LIN {X 0,Y 688.644,Z 762.06,A -85,B 0,C 180,E1 4140.007,E2 4140.007} C_VEL
LIN {X 0,Y 688.645,Z 762.06,A -85,B 0,C 180,E1 4145.042,E2 4145.042} C_VEL
LIN {X 0,Y 688.471,Z 762.06,A -85,B 0,C 180,E1 4150.119,E2 4150.119} C_VEL
LIN {X 0,Y 688.438,Z 762.06,A -85,B 0,C 180,E1 4155.277,E2 4155.277} C_VEL
LIN {X 0,Y 688.385,Z 762.06,A -85,B 0,C 180,E1 4160.05,E2 4160.05} C_VEL
LIN {X 0,Y 687.119,Z 762.06,A -85,B 0,C 180,E1 4160.769,E2 4160.769} C_VEL
LIN {X 0,Y 680.471,Z 762.06,A -85,B 0,C 180,E1 4162.723,E2 4162.723} C_VEL
LIN {X 0,Y 680.377,Z 762.06,A -85,B 0,C 180,E1 4162.908,E2 4162.908} C_VEL
LIN {X 0,Y 680.412,Z 762.06,A -85,B 0,C 180,E1 4167.804,E2 4167.804} C_VEL
LIN {X 0,Y 680.284,Z 762.06,A -85,B 0,C 180,E1 4172.424,E2 4172.424} C_VEL
LIN {X 0,Y 680.225,Z 762.06,A -85,B 0,C 180,E1 4176.894,E2 4176.894} C_VEL
LIN {X 0,Y 680.38,Z 762.06,A -85,B 0,C 180,E1 4182.867,E2 4182.867} C_VEL
LIN {X 0,Y 680.225,Z 762.06,A -85,B 0,C 180,E1 4188.271,E2 4188.271} C_VEL
LIN {X 0,Y 685.455,Z 772.734,A -85,B 0,C 180,E1 4188.863,E2 4188.863} C_VEL
LIN {X 0,Y 698.064,Z 795.344,A -85,B 0,C 180,E1 4190.059,E2 4190.059} C_VEL
LIN {X 0,Y 697.442,Z 854.76,A -85,B 0,C 180,E1 4190.981,E2 4190.981} C_VEL
LIN {X 0,Y 695.603,Z 898.868,A -85,B 0,C 180,E1 4192.105,E2 4192.105} C_VEL
LIN {X 0,Y 693.258,Z 948.265,A -85,B 0,C 180,E1 4193.947,E2 4193.947} C_VEL
LIN {X 0,Y 690.751,Z 992.677,A -85,B 0,C 180,E1 4196.173,E2 4196.173} C_VEL
LIN {X 0,Y 688.172,Z 1037.406,A -85,B 0,C 180,E1 4199.062,E2 4199.062} C_VEL
LIN {X 0,Y 685.781,Z 1076.683,A -85,B 0,C 180,E1 4202.265,E2 4202.265} C_VEL
LIN {X 0,Y 683.938,Z 1110.79,A -85,B 0,C 180,E1 4205.7,E2 4205.7} C_VEL
LIN {X 0,Y 682.434,Z 1142.324,A -85,B 0,C 180,E1 4209.682,E2 4209.682} C_VEL
LIN {X 0,Y 681.538,Z 1166.468,A -85,B 0,C 180,E1 4213.578,E2 4213.578} C_VEL
LIN {X 0,Y 681.033,Z 1185.03,A -85,B 0,C 180,E1 4217.501,E2 4217.501} C_VEL
LIN {X 0,Y 680.865,Z 1197.33,A -85,B 0,C 180,E1 4221.062,E2 4221.062} C_VEL
LIN {X 0,Y 680.767,Z 1205.91,A -85,B 0,C 180,E1 4224.905,E2 4224.905} C_VEL
LIN {X 0,Y 680.672,Z 1209.668,A -85,B 0,C 180,E1 4228.727,E2 4228.727} C_VEL
LIN {X 0,Y 680.871,Z 1208.953,A -85,B 0,C 180,E1 4232.543,E2 4232.543} C_VEL
LIN {X 0,Y 680.861,Z 1203.571,A -85,B 0,C 180,E1 4236.371,E2 4236.371} C_VEL
LIN {X 0,Y 681.018,Z 1192.319,A -85,B 0,C 180,E1 4240.547,E2 4240.547} C_VEL
LIN {X 0,Y 681.312,Z 1175.162,A -85,B 0,C 180,E1 4244.725,E2 4244.725} C_VEL
LIN {X 0,Y 682.005,Z 1153.941,A -85,B 0,C 180,E1 4248.572,E2 4248.572} C_VEL
LIN {X 0,Y 683.15,Z 1126.486,A -85,B 0,C 180,E1 4252.43,E2 4252.43} C_VEL
LIN {X 0,Y 684.773,Z 1094.478,A -85,B 0,C 180,E1 4256.038,E2 4256.038} C_VEL
LIN {X 0,Y 687.044,Z 1055.156,A -85,B 0,C 180,E1 4259.585,E2 4259.585} C_VEL
LIN {X 0,Y 689.594,Z 1013.392,A -85,B 0,C 180,E1 4262.572,E2 4262.572} C_VEL
LIN {X 0,Y 692.183,Z 970.786,A -85,B 0,C 180,E1 4264.995,E2 4264.995} C_VEL
LIN {X 0,Y 694.562,Z 925.309,A -85,B 0,C 180,E1 4266.975,E2 4266.975} C_VEL
LIN {X 0,Y 696.481,Z 879.014,A -85,B 0,C 180,E1 4268.46,E2 4268.46} C_VEL
LIN {X 0,Y 697.908,Z 831.825,A -85,B 0,C 180,E1 4269.439,E2 4269.439} C_VEL
LIN {X 0,Y 697.724,Z 794.961,A -85,B 0,C 180,E1 4269.969,E2 4269.969} C_VEL
LIN {X 0,Y 680.46,Z 763.676,A -85,B 0,C 180,E1 4271.63,E2 4271.63} C_VEL
LIN {X 0,Y 680.306,Z 762.06,A -85,B 0,C 180,E1 4271.725,E2 4271.725} C_VEL
LIN {X 0,Y 680.274,Z 762.06,A -85,B 0,C 180,E1 4276.476,E2 4276.476} C_VEL
LIN {X 0,Y 680.206,Z 762.06,A -85,B 0,C 180,E1 4281.532,E2 4281.532} C_VEL
LIN {X 0,Y 680.178,Z 762.06,A -85,B 0,C 180,E1 4286.257,E2 4286.257} C_VEL
LIN {X 0,Y 680.205,Z 762.06,A -85,B 0,C 180,E1 4290.738,E2 4290.738} C_VEL
LIN {X 0,Y 680.287,Z 762.06,A -85,B 0,C 180,E1 4295.604,E2 4295.604} C_VEL
LIN {X 0,Y 680.322,Z 762.06,A -85,B 0,C 180,E1 4300.533,E2 4300.533} C_VEL
LIN {X 0,Y 680.504,Z 762.06,A -85,B 0,C 180,E1 4304.54,E2 4304.54} C_VEL
LIN {X 0,Y 680.545,Z 762.06,A -85,B 0,C 180,E1 4309.762,E2 4309.762} C_VEL
LIN {X 0,Y 680.769,Z 762.06,A -85,B 0,C 180,E1 4314.899,E2 4314.899} C_VEL
LIN {X 0,Y 680.714,Z 762.06,A -85,B 0,C 180,E1 4319.993,E2 4319.993} C_VEL
LIN {X 0,Y 680.699,Z 762.06,A -85,B 0,C 180,E1 4325.086,E2 4325.086} C_VEL
LIN {X 0,Y 680.588,Z 762.06,A -85,B 0,C 180,E1 4330.223,E2 4330.223} C_VEL
LIN {X 0,Y 680.249,Z 762.06,A -85,B 0,C 180,E1 4335.451,E2 4335.451} C_VEL
LIN {X 0,Y 680.284,Z 762.06,A -85,B 0,C 180,E1 4341.103,E2 4341.103} C_VEL
LIN {X 0,Y 680.228,Z 762.06,A -85,B 0,C 180,E1 4346.366,E2 4346.366} C_VEL
LIN {X 0,Y 680.227,Z 762.06,A -85,B 0,C 180,E1 4350.714,E2 4350.714} C_VEL
LIN {X 0,Y 680.253,Z 762.06,A -85,B 0,C 180,E1 4355.265,E2 4355.265} C_VEL
LIN {X 0,Y 680.097,Z 762.06,A -85,B 0,C 180,E1 4360.101,E2 4360.101} C_VEL
LIN {X 0,Y 680.121,Z 762.06,A -85,B 0,C 180,E1 4365.297,E2 4365.297} C_VEL
LIN {X 0,Y 680.444,Z 762.06,A -85,B 0,C 180,E1 4368.694,E2 4368.694} C_VEL
LIN {X 0,Y 684.939,Z 771.765,A -85,B 0,C 180,E1 4369.176,E2 4369.176} C_VEL
LIN {X 0,Y 698.059,Z 795.739,A -85,B 0,C 180,E1 4370.431,E2 4370.431} C_VEL
LIN {X 0,Y 696.879,Z 840.886,A -85,B 0,C 180,E1 4371.297,E2 4371.297} C_VEL
LIN {X 0,Y 694.891,Z 887.195,A -85,B 0,C 180,E1 4372.674,E2 4372.674} C_VEL
LIN {X 0,Y 692.53,Z 933.533,A -85,B 0,C 180,E1 4374.61,E2 4374.61} C_VEL
LIN {X 0,Y 689.958,Z 977.454,A -85,B 0,C 180,E1 4377.004,E2 4377.004} C_VEL
LIN {X 0,Y 687.283,Z 1021.111,A -85,B 0,C 180,E1 4380.054,E2 4380.054} C_VEL
LIN {X 0,Y 685.096,Z 1057.631,A -85,B 0,C 180,E1 4383.243,E2 4383.243} C_VEL
LIN {X 0,Y 683.355,Z 1091.448,A -85,B 0,C 180,E1 4386.89,E2 4386.89} C_VEL
LIN {X 0,Y 682.041,Z 1119.879,A -85,B 0,C 180,E1 4390.758,E2 4390.758} C_VEL
LIN {X 0,Y 681.336,Z 1141.96,A -85,B 0,C 180,E1 4394.566,E2 4394.566} C_VEL
LIN {X 0,Y 680.908,Z 1159.052,A -85,B 0,C 180,E1 4398.479,E2 4398.479} C_VEL
LIN {X 0,Y 680.788,Z 1170.831,A -85,B 0,C 180,E1 4402.347,E2 4402.347} C_VEL
LIN {X 0,Y 680.711,Z 1177.734,A -85,B 0,C 180,E1 4406.182,E2 4406.182} C_VEL
LIN {X 0,Y 680.653,Z 1179.995,A -85,B 0,C 180,E1 4410.001,E2 4410.001} C_VEL
LIN {X 0,Y 680.788,Z 1177.623,A -85,B 0,C 180,E1 4413.819,E2 4413.819} C_VEL
LIN {X 0,Y 680.868,Z 1170.609,A -85,B 0,C 180,E1 4417.653,E2 4417.653} C_VEL
LIN {X 0,Y 681.084,Z 1157.714,A -85,B 0,C 180,E1 4421.788,E2 4421.788} C_VEL
LIN {X 0,Y 681.543,Z 1139.745,A -85,B 0,C 180,E1 4425.761,E2 4425.761} C_VEL
LIN {X 0,Y 682.329,Z 1116.346,A -85,B 0,C 180,E1 4429.684,E2 4429.684} C_VEL
LIN {X 0,Y 683.528,Z 1087.766,A -85,B 0,C 180,E1 4433.45,E2 4433.45} C_VEL
LIN {X 0,Y 685.418,Z 1053.408,A -85,B 0,C 180,E1 4437.079,E2 4437.079} C_VEL
LIN {X 0,Y 687.672,Z 1014.547,A -85,B 0,C 180,E1 4440.359,E2 4440.359} C_VEL
LIN {X 0,Y 690.172,Z 974.441,A -85,B 0,C 180,E1 4443.088,E2 4443.088} C_VEL
LIN {X 0,Y 692.75,Z 929.374,A -85,B 0,C 180,E1 4445.498,E2 4445.498} C_VEL
LIN {X 0,Y 694.997,Z 883.395,A -85,B 0,C 180,E1 4447.375,E2 4447.375} C_VEL
LIN {X 0,Y 696.946,Z 833.509,A -85,B 0,C 180,E1 4448.795,E2 4448.795} C_VEL
LIN {X 0,Y 697.575,Z 794.939,A -85,B 0,C 180,E1 4449.524,E2 4449.524} C_VEL
LIN {X 0,Y 680.312,Z 763.034,A -85,B 0,C 180,E1 4451.191,E2 4451.191} C_VEL
LIN {X 0,Y 680.293,Z 762.06,A -85,B 0,C 180,E1 4451.404,E2 4451.404} C_VEL
LIN {X 0,Y 680.207,Z 762.06,A -85,B 0,C 180,E1 4456.491,E2 4456.491} C_VEL
LIN {X 0,Y 680.193,Z 762.06,A -85,B 0,C 180,E1 4461.55,E2 4461.55} C_VEL
LIN {X 0,Y 680.163,Z 762.06,A -85,B 0,C 180,E1 4466.274,E2 4466.274} C_VEL
LIN {X 0,Y 680.147,Z 762.06,A -85,B 0,C 180,E1 4470.752,E2 4470.752} C_VEL
LIN {X 0,Y 680.156,Z 762.06,A -85,B 0,C 180,E1 4475.632,E2 4475.632} C_VEL
LIN {X 0,Y 680.195,Z 762.06,A -85,B 0,C 180,E1 4480.545,E2 4480.545} C_VEL
LIN {X 0,Y 680.372,Z 762.06,A -85,B 0,C 180,E1 4485.868,E2 4485.868} C_VEL
LIN {X 0,Y 680.583,Z 762.06,A -85,B 0,C 180,E1 4491.067,E2 4491.067} C_VEL
LIN {X 0,Y 680.735,Z 762.06,A -85,B 0,C 180,E1 4496.189,E2 4496.189} C_VEL
LIN {X 0,Y 680.877,Z 762.06,A -85,B 0,C 180,E1 4501.279,E2 4501.279} C_VEL
LIN {X 0,Y 680.553,Z 762.06,A -85,B 0,C 180,E1 4506.381,E2 4506.381} C_VEL
LIN {X 0,Y 680.516,Z 762.06,A -85,B 0,C 180,E1 4511.534,E2 4511.534} C_VEL
LIN {X 0,Y 680.578,Z 762.06,A -85,B 0,C 180,E1 4516.782,E2 4516.782} C_VEL
LIN {X 0,Y 680.436,Z 762.06,A -85,B 0,C 180,E1 4522.186,E2 4522.186} C_VEL
LIN {X 0,Y 680.377,Z 762.06,A -85,B 0,C 180,E1 4522.908,E2 4522.908} C_VEL
LIN {X 0,Y 676.412,Z 762.06,A -85,B 0,C 180,E1 4524.341,E2 4524.341} C_VEL
LIN {X 0,Y 672.447,Z 762.06,A -85,B 0,C 180,E1 4525.791,E2 4525.791} C_VEL
LIN {X 0,Y 672.369,Z 762.06,A -85,B 0,C 180,E1 4531.13,E2 4531.13} C_VEL
LIN {X 0,Y 672.305,Z 762.06,A -85,B 0,C 180,E1 4535.985,E2 4535.985} C_VEL
LIN {X 0,Y 672.273,Z 762.06,A -85,B 0,C 180,E1 4540.685,E2 4540.685} C_VEL
LIN {X 0,Y 672.385,Z 762.06,A -85,B 0,C 180,E1 4545.837,E2 4545.837} C_VEL
LIN {X 0,Y 672.303,Z 762.06,A -85,B 0,C 180,E1 4547.718,E2 4547.718} C_VEL
LIN {X 0,Y 674.702,Z 767.723,A -85,B 0,C 180,E1 4547.991,E2 4547.991} C_VEL
LIN {X 0,Y 691.939,Z 798.188,A -85,B 0,C 180,E1 4549.671,E2 4549.671} C_VEL
LIN {X 0,Y 691.267,Z 855.727,A -85,B 0,C 180,E1 4550.587,E2 4550.587} C_VEL
LIN {X 0,Y 689.185,Z 900.544,A -85,B 0,C 180,E1 4551.748,E2 4551.748} C_VEL
LIN {X 0,Y 686.622,Z 950.179,A -85,B 0,C 180,E1 4553.631,E2 4553.631} C_VEL
LIN {X 0,Y 683.749,Z 995.548,A -85,B 0,C 180,E1 4555.958,E2 4555.958} C_VEL
LIN {X 0,Y 681.033,Z 1038.439,A -85,B 0,C 180,E1 4558.778,E2 4558.778} C_VEL
LIN {X 0,Y 678.354,Z 1078.521,A -85,B 0,C 180,E1 4562.108,E2 4562.108} C_VEL
LIN {X 0,Y 676.326,Z 1112.265,A -85,B 0,C 180,E1 4565.584,E2 4565.584} C_VEL
LIN {X 0,Y 674.716,Z 1142.775,A -85,B 0,C 180,E1 4569.504,E2 4569.504} C_VEL
LIN {X 0,Y 673.749,Z 1166.47,A -85,B 0,C 180,E1 4573.383,E2 4573.383} C_VEL
LIN {X 0,Y 673.235,Z 1183.698,A -85,B 0,C 180,E1 4577.029,E2 4577.029} C_VEL
LIN {X 0,Y 672.995,Z 1197.33,A -85,B 0,C 180,E1 4580.956,E2 4580.956} C_VEL
LIN {X 0,Y 672.869,Z 1205.909,A -85,B 0,C 180,E1 4584.845,E2 4584.845} C_VEL
LIN {X 0,Y 672.784,Z 1209.668,A -85,B 0,C 180,E1 4588.712,E2 4588.712} C_VEL
LIN {X 0,Y 672.989,Z 1208.95,A -85,B 0,C 180,E1 4592.573,E2 4592.573} C_VEL
LIN {X 0,Y 672.964,Z 1203.571,A -85,B 0,C 180,E1 4596.446,E2 4596.446} C_VEL
LIN {X 0,Y 673.144,Z 1192.318,A -85,B 0,C 180,E1 4600.672,E2 4600.672} C_VEL
LIN {X 0,Y 673.45,Z 1175.789,A -85,B 0,C 180,E1 4604.767,E2 4604.767} C_VEL
LIN {X 0,Y 674.199,Z 1154.981,A -85,B 0,C 180,E1 4608.625,E2 4608.625} C_VEL
LIN {X 0,Y 675.447,Z 1128.012,A -85,B 0,C 180,E1 4612.503,E2 4612.503} C_VEL
LIN {X 0,Y 677.242,Z 1096.462,A -85,B 0,C 180,E1 4616.146,E2 4616.146} C_VEL
LIN {X 0,Y 679.636,Z 1058.656,A -85,B 0,C 180,E1 4619.634,E2 4619.634} C_VEL
LIN {X 0,Y 682.239,Z 1019.824,A -85,B 0,C 180,E1 4622.526,E2 4622.526} C_VEL
LIN {X 0,Y 685.072,Z 976.814,A -85,B 0,C 180,E1 4625.071,E2 4625.071} C_VEL
LIN {X 0,Y 687.758,Z 931.735,A -85,B 0,C 180,E1 4627.138,E2 4627.138} C_VEL
LIN {X 0,Y 690.086,Z 882.336,A -85,B 0,C 180,E1 4628.782,E2 4628.782} C_VEL
LIN {X 0,Y 691.719,Z 834.798,A -85,B 0,C 180,E1 4629.812,E2 4629.812} C_VEL
LIN {X 0,Y 691.594,Z 797.998,A -85,B 0,C 180,E1 4630.356,E2 4630.356} C_VEL
LIN {X 0,Y 672.459,Z 763.065,A -85,B 0,C 180,E1 4632.248,E2 4632.248} C_VEL
LIN {X 0,Y 672.43,Z 762.06,A -85,B 0,C 180,E1 4632.389,E2 4632.389} C_VEL
LIN {X 0,Y 672.29,Z 762.06,A -85,B 0,C 180,E1 4637.879,E2 4637.879} C_VEL
LIN {X 0,Y 672.265,Z 762.06,A -85,B 0,C 180,E1 4642.63,E2 4642.63} C_VEL
LIN {X 0,Y 672.248,Z 762.06,A -85,B 0,C 180,E1 4647.347,E2 4647.347} C_VEL
LIN {X 0,Y 672.294,Z 762.06,A -85,B 0,C 180,E1 4651.83,E2 4651.83} C_VEL
LIN {X 0,Y 672.32,Z 762.06,A -85,B 0,C 180,E1 4657.148,E2 4657.148} C_VEL
LIN {X 0,Y 672.451,Z 762.06,A -85,B 0,C 180,E1 4661.658,E2 4661.658} C_VEL
LIN {X 0,Y 672.619,Z 762.06,A -85,B 0,C 180,E1 4667.011,E2 4667.011} C_VEL
LIN {X 0,Y 672.659,Z 762.06,A -85,B 0,C 180,E1 4672.247,E2 4672.247} C_VEL
LIN {X 0,Y 672.783,Z 762.06,A -85,B 0,C 180,E1 4676.129,E2 4676.129} C_VEL
LIN {X 0,Y 672.819,Z 762.06,A -85,B 0,C 180,E1 4679.993,E2 4679.993} C_VEL
LIN {X 0,Y 672.791,Z 762.06,A -85,B 0,C 180,E1 4685.146,E2 4685.146} C_VEL
LIN {X 0,Y 672.686,Z 762.06,A -85,B 0,C 180,E1 4690.344,E2 4690.344} C_VEL
LIN {X 0,Y 672.328,Z 762.06,A -85,B 0,C 180,E1 4695.637,E2 4695.637} C_VEL
LIN {X 0,Y 672.394,Z 762.06,A -85,B 0,C 180,E1 4701.063,E2 4701.063} C_VEL
LIN {X 0,Y 672.329,Z 762.06,A -85,B 0,C 180,E1 4705.971,E2 4705.971} C_VEL
LIN {X 0,Y 672.283,Z 762.06,A -85,B 0,C 180,E1 4711.337,E2 4711.337} C_VEL
LIN {X 0,Y 672.29,Z 762.06,A -85,B 0,C 180,E1 4715.986,E2 4715.986} C_VEL
LIN {X 0,Y 672.178,Z 762.06,A -85,B 0,C 180,E1 4720.672,E2 4720.672} C_VEL
LIN {X 0,Y 672.247,Z 762.06,A -85,B 0,C 180,E1 4725.98,E2 4725.98} C_VEL
LIN {X 0,Y 672.509,Z 762.298,A -85,B 0,C 180,E1 4728.123,E2 4728.123} C_VEL
LIN {X 0,Y 677.269,Z 772.18,A -85,B 0,C 180,E1 4728.619,E2 4728.619} C_VEL
LIN {X 0,Y 691.7,Z 798.296,A -85,B 0,C 180,E1 4730.036,E2 4730.036} C_VEL
LIN {X 0,Y 690.549,Z 845.158,A -85,B 0,C 180,E1 4730.991,E2 4730.991} C_VEL
LIN {X 0,Y 688.289,Z 891.147,A -85,B 0,C 180,E1 4732.416,E2 4732.416} C_VEL
LIN {X 0,Y 685.728,Z 936.838,A -85,B 0,C 180,E1 4734.377,E2 4734.377} C_VEL
LIN {X 0,Y 682.976,Z 978.386,A -85,B 0,C 180,E1 4736.687,E2 4736.687} C_VEL
LIN {X 0,Y 680.09,Z 1021.741,A -85,B 0,C 180,E1 4739.756,E2 4739.756} C_VEL
LIN {X 0,Y 677.704,Z 1057.859,A -85,B 0,C 180,E1 4742.951,E2 4742.951} C_VEL
LIN {X 0,Y 675.765,Z 1090.729,A -85,B 0,C 180,E1 4746.53,E2 4746.53} C_VEL
LIN {X 0,Y 674.42,Z 1117.652,A -85,B 0,C 180,E1 4750.188,E2 4750.188} C_VEL
LIN {X 0,Y 673.577,Z 1140.221,A -85,B 0,C 180,E1 4754.049,E2 4754.049} C_VEL
LIN {X 0,Y 673.128,Z 1157.29,A -85,B 0,C 180,E1 4757.865,E2 4757.865} C_VEL
LIN {X 0,Y 672.921,Z 1169.284,A -85,B 0,C 180,E1 4761.633,E2 4761.633} C_VEL
LIN {X 0,Y 672.824,Z 1175.978,A -85,B 0,C 180,E1 4764.846,E2 4764.846} C_VEL
LIN {X 0,Y 672.757,Z 1179.681,A -85,B 0,C 180,E1 4768.714,E2 4768.714} C_VEL
LIN {X 0,Y 672.798,Z 1178.913,A -85,B 0,C 180,E1 4772.575,E2 4772.575} C_VEL
LIN {X 0,Y 672.87,Z 1173.478,A -85,B 0,C 180,E1 4776.448,E2 4776.448} C_VEL
LIN {X 0,Y 672.999,Z 1163.27,A -85,B 0,C 180,E1 4780.349,E2 4780.349} C_VEL
LIN {X 0,Y 673.396,Z 1147.805,A -85,B 0,C 180,E1 4784.291,E2 4784.291} C_VEL
LIN {X 0,Y 674.097,Z 1126.687,A -85,B 0,C 180,E1 4788.291,E2 4788.291} C_VEL
LIN {X 0,Y 675.278,Z 1100.873,A -85,B 0,C 180,E1 4792.091,E2 4792.091} C_VEL
LIN {X 0,Y 677.187,Z 1067.641,A -85,B 0,C 180,E1 4795.975,E2 4795.975} C_VEL
LIN {X 0,Y 679.363,Z 1032.13,A -85,B 0,C 180,E1 4799.298,E2 4799.298} C_VEL
LIN {X 0,Y 682.103,Z 991.874,A -85,B 0,C 180,E1 4802.348,E2 4802.348} C_VEL
LIN {X 0,Y 684.936,Z 947.358,A -85,B 0,C 180,E1 4805.003,E2 4805.003} C_VEL
LIN {X 0,Y 687.815,Z 901.798,A -85,B 0,C 180,E1 4807.087,E2 4807.087} C_VEL
LIN {X 0,Y 689.944,Z 857.888,A -85,B 0,C 180,E1 4808.576,E2 4808.576} C_VEL
LIN {X 0,Y 691.564,Z 815.02,A -85,B 0,C 180,E1 4809.575,E2 4809.575} C_VEL
LIN {X 0,Y 691.423,Z 797.904,A -85,B 0,C 180,E1 4809.9,E2 4809.9} C_VEL
LIN {X 0,Y 672.516,Z 763.039,A -85,B 0,C 180,E1 4811.776,E2 4811.776} C_VEL
LIN {X 0,Y 672.453,Z 762.06,A -85,B 0,C 180,E1 4811.875,E2 4811.875} C_VEL
LIN {X 0,Y 672.335,Z 762.06,A -85,B 0,C 180,E1 4815.991,E2 4815.991} C_VEL
LIN {X 0,Y 672.306,Z 762.06,A -85,B 0,C 180,E1 4821.014,E2 4821.014} C_VEL
LIN {X 0,Y 672.267,Z 762.06,A -85,B 0,C 180,E1 4826.273,E2 4826.273} C_VEL
LIN {X 0,Y 672.232,Z 762.06,A -85,B 0,C 180,E1 4831.844,E2 4831.844} C_VEL
LIN {X 0,Y 672.186,Z 762.06,A -85,B 0,C 180,E1 4837.178,E2 4837.178} C_VEL
LIN {X 0,Y 672.188,Z 762.06,A -85,B 0,C 180,E1 4841.666,E2 4841.666} C_VEL
LIN {X 0,Y 672.471,Z 762.06,A -85,B 0,C 180,E1 4847.023,E2 4847.023} C_VEL
LIN {X 0,Y 672.764,Z 762.06,A -85,B 0,C 180,E1 4852.263,E2 4852.263} C_VEL
LIN {X 0,Y 672.897,Z 762.06,A -85,B 0,C 180,E1 4857.434,E2 4857.434} C_VEL
LIN {X 0,Y 672.742,Z 762.06,A -85,B 0,C 180,E1 4862.582,E2 4862.582} C_VEL
LIN {X 0,Y 672.646,Z 762.06,A -85,B 0,C 180,E1 4866.456,E2 4866.456} C_VEL
LIN {X 0,Y 672.615,Z 762.06,A -85,B 0,C 180,E1 4871.672,E2 4871.672} C_VEL
LIN {X 0,Y 672.672,Z 762.06,A -85,B 0,C 180,E1 4876.985,E2 4876.985} C_VEL
LIN {X 0,Y 672.502,Z 762.06,A -85,B 0,C 180,E1 4882.462,E2 4882.462} C_VEL
LIN {X 0,Y 672.447,Z 762.06,A -85,B 0,C 180,E1 4885.791,E2 4885.791} C_VEL
LIN {X 0,Y 668.538,Z 762.06,A -85,B 0,C 180,E1 4887.249,E2 4887.249} C_VEL
LIN {X 0,Y 664.492,Z 762.06,A -85,B 0,C 180,E1 4888.723,E2 4888.723} C_VEL
LIN {X 0,Y 664.477,Z 762.06,A -85,B 0,C 180,E1 4893.083,E2 4893.083} C_VEL
LIN {X 0,Y 664.339,Z 762.06,A -85,B 0,C 180,E1 4897.894,E2 4897.894} C_VEL
LIN {X 0,Y 664.493,Z 762.06,A -85,B 0,C 180,E1 4903.305,E2 4903.305} C_VEL
LIN {X 0,Y 664.371,Z 762.211,A -85,B 0,C 180,E1 4907.103,E2 4907.103} C_VEL
LIN {X 0,Y 666.964,Z 767.901,A -85,B 0,C 180,E1 4907.391,E2 4907.391} C_VEL
LIN {X 0,Y 686.062,Z 801.684,A -85,B 0,C 180,E1 4909.3,E2 4909.3} C_VEL
LIN {X 0,Y 685.061,Z 857.199,A -85,B 0,C 180,E1 4910.195,E2 4910.195} C_VEL
LIN {X 0,Y 682.88,Z 901.201,A -85,B 0,C 180,E1 4911.354,E2 4911.354} C_VEL
LIN {X 0,Y 680.145,Z 950.226,A -85,B 0,C 180,E1 4913.23,E2 4913.23} C_VEL
LIN {X 0,Y 677.107,Z 994.163,A -85,B 0,C 180,E1 4915.49,E2 4915.49} C_VEL
LIN {X 0,Y 674.057,Z 1037.191,A -85,B 0,C 180,E1 4918.324,E2 4918.324} C_VEL
LIN {X 0,Y 671.185,Z 1075.891,A -85,B 0,C 180,E1 4921.532,E2 4921.532} C_VEL
LIN {X 0,Y 668.935,Z 1109.424,A -85,B 0,C 180,E1 4924.954,E2 4924.954} C_VEL
LIN {X 0,Y 667.132,Z 1140.454,A -85,B 0,C 180,E1 4928.925,E2 4928.925} C_VEL
LIN {X 0,Y 666.104,Z 1164.713,A -85,B 0,C 180,E1 4932.847,E2 4932.847} C_VEL
LIN {X 0,Y 665.396,Z 1183.699,A -85,B 0,C 180,E1 4936.873,E2 4936.873} C_VEL
LIN {X 0,Y 665.11,Z 1197.33,A -85,B 0,C 180,E1 4940.848,E2 4940.848} C_VEL
LIN {X 0,Y 665.001,Z 1205.909,A -85,B 0,C 180,E1 4944.784,E2 4944.784} C_VEL
LIN {X 0,Y 664.903,Z 1209.668,A -85,B 0,C 180,E1 4948.697,E2 4948.697} C_VEL
LIN {X 0,Y 665.111,Z 1208.947,A -85,B 0,C 180,E1 4952.604,E2 4952.604} C_VEL
LIN {X 0,Y 665.065,Z 1203.571,A -85,B 0,C 180,E1 4956.523,E2 4956.523} C_VEL
LIN {X 0,Y 665.269,Z 1192.318,A -85,B 0,C 180,E1 4960.8,E2 4960.8} C_VEL
LIN {X 0,Y 665.615,Z 1176.042,A -85,B 0,C 180,E1 4964.89,E2 4964.89} C_VEL
LIN {X 0,Y 666.406,Z 1154.983,A -85,B 0,C 180,E1 4968.851,E2 4968.851} C_VEL
LIN {X 0,Y 667.757,Z 1128.129,A -85,B 0,C 180,E1 4972.761,E2 4972.761} C_VEL
LIN {X 0,Y 669.807,Z 1096.461,A -85,B 0,C 180,E1 4976.459,E2 4976.459} C_VEL
LIN {X 0,Y 672.407,Z 1058.655,A -85,B 0,C 180,E1 4979.985,E2 4979.985} C_VEL
LIN {X 0,Y 675.293,Z 1019.826,A -85,B 0,C 180,E1 4982.903,E2 4982.903} C_VEL
LIN {X 0,Y 678.381,Z 976.811,A -85,B 0,C 180,E1 4985.469,E2 4985.469} C_VEL
LIN {X 0,Y 681.29,Z 932.908,A -85,B 0,C 180,E1 4987.503,E2 4987.503} C_VEL
LIN {X 0,Y 683.71,Z 884.987,A -85,B 0,C 180,E1 4989.129,E2 4989.129} C_VEL
LIN {X 0,Y 685.583,Z 836.827,A -85,B 0,C 180,E1 4990.203,E2 4990.203} C_VEL
LIN {X 0,Y 685.716,Z 801.552,A -85,B 0,C 180,E1 4990.726,E2 4990.726} C_VEL
LIN {X 0,Y 664.644,Z 763.546,A -85,B 0,C 180,E1 4992.856,E2 4992.856} C_VEL
LIN {X 0,Y 664.489,Z 762.06,A -85,B 0,C 180,E1 4992.929,E2 4992.929} C_VEL
LIN {X 0,Y 664.362,Z 762.06,A -85,B 0,C 180,E1 4996.968,E2 4996.968} C_VEL
LIN {X 0,Y 664.356,Z 762.06,A -85,B 0,C 180,E1 5002.107,E2 5002.107} C_VEL
LIN {X 0,Y 664.354,Z 762.06,A -85,B 0,C 180,E1 5007.307,E2 5007.307} C_VEL
LIN {X 0,Y 664.392,Z 762.06,A -85,B 0,C 180,E1 5012.938,E2 5012.938} C_VEL
LIN {X 0,Y 664.439,Z 762.06,A -85,B 0,C 180,E1 5017.25,E2 5017.25} C_VEL
LIN {X 0,Y 664.666,Z 762.06,A -85,B 0,C 180,E1 5022.804,E2 5022.804} C_VEL
LIN {X 0,Y 664.691,Z 762.06,A -85,B 0,C 180,E1 5028.187,E2 5028.187} C_VEL
LIN {X 0,Y 664.739,Z 762.06,A -85,B 0,C 180,E1 5033.467,E2 5033.467} C_VEL
LIN {X 0,Y 665.055,Z 762.06,A -85,B 0,C 180,E1 5038.691,E2 5038.691} C_VEL
LIN {X 0,Y 664.931,Z 762.06,A -85,B 0,C 180,E1 5043.901,E2 5043.901} C_VEL
LIN {X 0,Y 664.746,Z 762.06,A -85,B 0,C 180,E1 5049.147,E2 5049.147} C_VEL
LIN {X 0,Y 664.511,Z 762.06,A -85,B 0,C 180,E1 5054.476,E2 5054.476} C_VEL
LIN {X 0,Y 664.42,Z 762.06,A -85,B 0,C 180,E1 5059.936,E2 5059.936} C_VEL
LIN {X 0,Y 664.44,Z 762.06,A -85,B 0,C 180,E1 5064.537,E2 5064.537} C_VEL
LIN {X 0,Y 664.361,Z 762.06,A -85,B 0,C 180,E1 5070.196,E2 5070.196} C_VEL
LIN {X 0,Y 664.374,Z 762.06,A -85,B 0,C 180,E1 5075.035,E2 5075.035} C_VEL
LIN {X 0,Y 664.297,Z 762.06,A -85,B 0,C 180,E1 5079.548,E2 5079.548} C_VEL
LIN {X 0,Y 664.249,Z 762.06,A -85,B 0,C 180,E1 5085.153,E2 5085.153} C_VEL
LIN {X 0,Y 664.507,Z 762.118,A -85,B 0,C 180,E1 5087.5,E2 5087.5} C_VEL
LIN {X 0,Y 666.912,Z 767.711,A -85,B 0,C 180,E1 5087.768,E2 5087.768} C_VEL
LIN {X 0,Y 685.678,Z 801.447,A -85,B 0,C 180,E1 5089.664,E2 5089.664} C_VEL
LIN {X 0,Y 684.295,Z 846.863,A -85,B 0,C 180,E1 5090.616,E2 5090.616} C_VEL
LIN {X 0,Y 681.831,Z 892.603,A -85,B 0,C 180,E1 5092.058,E2 5092.058} C_VEL
LIN {X 0,Y 679.13,Z 936.661,A -85,B 0,C 180,E1 5093.968,E2 5093.968} C_VEL
LIN {X 0,Y 676.026,Z 979.31,A -85,B 0,C 180,E1 5096.364,E2 5096.364} C_VEL
LIN {X 0,Y 672.905,Z 1022.012,A -85,B 0,C 180,E1 5099.421,E2 5099.421} C_VEL
LIN {X 0,Y 670.21,Z 1059.406,A -85,B 0,C 180,E1 5102.784,E2 5102.784} C_VEL
LIN {X 0,Y 668.137,Z 1091.891,A -85,B 0,C 180,E1 5106.389,E2 5106.389} C_VEL
LIN {X 0,Y 666.589,Z 1119.875,A -85,B 0,C 180,E1 5110.294,E2 5110.294} C_VEL
LIN {X 0,Y 665.703,Z 1141.951,A -85,B 0,C 180,E1 5114.194,E2 5114.194} C_VEL
LIN {X 0,Y 665.187,Z 1159.049,A -85,B 0,C 180,E1 5118.203,E2 5118.203} C_VEL
LIN {X 0,Y 664.993,Z 1170.823,A -85,B 0,C 180,E1 5122.164,E2 5122.164} C_VEL
LIN {X 0,Y 664.917,Z 1177.732,A -85,B 0,C 180,E1 5126.091,E2 5126.091} C_VEL
LIN {X 0,Y 664.864,Z 1179.995,A -85,B 0,C 180,E1 5130.001,E2 5130.001} C_VEL
LIN {X 0,Y 665.014,Z 1177.624,A -85,B 0,C 180,E1 5133.909,E2 5133.909} C_VEL
LIN {X 0,Y 665.089,Z 1170.606,A -85,B 0,C 180,E1 5137.836,E2 5137.836} C_VEL
LIN {X 0,Y 665.38,Z 1157.437,A -85,B 0,C 180,E1 5142.148,E2 5142.148} C_VEL
LIN {X 0,Y 665.825,Z 1139.751,A -85,B 0,C 180,E1 5146.143,E2 5146.143} C_VEL
LIN {X 0,Y 666.861,Z 1115.311,A -85,B 0,C 180,E1 5150.325,E2 5150.325} C_VEL
LIN {X 0,Y 668.511,Z 1086.314,A -85,B 0,C 180,E1 5154.187,E2 5154.187} C_VEL
LIN {X 0,Y 670.805,Z 1052.018,A -85,B 0,C 180,E1 5157.855,E2 5157.855} C_VEL
LIN {X 0,Y 673.769,Z 1011.047,A -85,B 0,C 180,E1 5161.341,E2 5161.341} C_VEL
LIN {X 0,Y 676.715,Z 970.954,A -85,B 0,C 180,E1 5164.057,E2 5164.057} C_VEL
LIN {X 0,Y 679.784,Z 926.313,A -85,B 0,C 180,E1 5166.442,E2 5166.442} C_VEL
LIN {X 0,Y 682.415,Z 881.393,A -85,B 0,C 180,E1 5168.261,E2 5168.261} C_VEL
LIN {X 0,Y 684.677,Z 832.573,A -85,B 0,C 180,E1 5169.65,E2 5169.65} C_VEL
LIN {X 0,Y 685.458,Z 801.452,A -85,B 0,C 180,E1 5170.261,E2 5170.261} C_VEL
LIN {X 0,Y 664.7,Z 763.565,A -85,B 0,C 180,E1 5172.374,E2 5172.374} C_VEL
LIN {X 0,Y 664.554,Z 762.06,A -85,B 0,C 180,E1 5172.449,E2 5172.449} C_VEL
LIN {X 0,Y 664.303,Z 762.06,A -85,B 0,C 180,E1 5176.984,E2 5176.984} C_VEL
LIN {X 0,Y 664.346,Z 762.06,A -85,B 0,C 180,E1 5182.126,E2 5182.126} C_VEL
LIN {X 0,Y 664.337,Z 762.06,A -85,B 0,C 180,E1 5187.311,E2 5187.311} C_VEL
LIN {X 0,Y 664.326,Z 762.06,A -85,B 0,C 180,E1 5192.952,E2 5192.952} C_VEL
LIN {X 0,Y 664.394,Z 762.06,A -85,B 0,C 180,E1 5198.671,E2 5198.671} C_VEL
LIN {X 0,Y 664.409,Z 762.06,A -85,B 0,C 180,E1 5204.172,E2 5204.172} C_VEL
LIN {X 0,Y 664.777,Z 762.06,A -85,B 0,C 180,E1 5209.532,E2 5209.532} C_VEL
LIN {X 0,Y 664.814,Z 762.06,A -85,B 0,C 180,E1 5214.792,E2 5214.792} C_VEL
LIN {X 0,Y 664.969,Z 762.06,A -85,B 0,C 180,E1 5220.008,E2 5220.008} C_VEL
LIN {X 0,Y 664.934,Z 762.06,A -85,B 0,C 180,E1 5225.222,E2 5225.222} C_VEL
LIN {X 0,Y 664.742,Z 762.06,A -85,B 0,C 180,E1 5230.484,E2 5230.484} C_VEL
LIN {X 0,Y 664.699,Z 762.06,A -85,B 0,C 180,E1 5235.837,E2 5235.837} C_VEL
LIN {X 0,Y 664.652,Z 762.06,A -85,B 0,C 180,E1 5241.226,E2 5241.226} C_VEL
LIN {X 0,Y 664.545,Z 762.06,A -85,B 0,C 180,E1 5245.783,E2 5245.783} C_VEL
LIN {X 0,Y 664.492,Z 762.06,A -85,B 0,C 180,E1 5248.723,E2 5248.723} C_VEL
LIN {X 0,Y 660.489,Z 762.06,A -85,B 0,C 180,E1 5250.198,E2 5250.198} C_VEL
LIN {X 0,Y 656.553,Z 762.06,A -85,B 0,C 180,E1 5251.69,E2 5251.69} C_VEL
LIN {X 0,Y 656.462,Z 762.06,A -85,B 0,C 180,E1 5256.766,E2 5256.766} C_VEL
LIN {X 0,Y 656.518,Z 762.06,A -85,B 0,C 180,E1 5262.561,E2 5262.561} C_VEL
LIN {X 0,Y 656.464,Z 762.191,A -85,B 0,C 180,E1 5266.458,E2 5266.458} C_VEL
LIN {X 0,Y 658.905,Z 767.757,A -85,B 0,C 180,E1 5266.741,E2 5266.741} C_VEL
LIN {X 0,Y 680.093,Z 805.309,A -85,B 0,C 180,E1 5268.916,E2 5268.916} C_VEL
LIN {X 0,Y 678.893,Z 858.644,A -85,B 0,C 180,E1 5269.796,E2 5269.796} C_VEL
LIN {X 0,Y 676.484,Z 903.636,A -85,B 0,C 180,E1 5271.01,E2 5271.01} C_VEL
LIN {X 0,Y 673.529,Z 952.182,A -85,B 0,C 180,E1 5272.902,E2 5272.902} C_VEL
LIN {X 0,Y 670.079,Z 997.78,A -85,B 0,C 180,E1 5275.308,E2 5275.308} C_VEL
LIN {X 0,Y 666.849,Z 1039.766,A -85,B 0,C 180,E1 5278.144,E2 5278.144} C_VEL
LIN {X 0,Y 663.606,Z 1080.436,A -85,B 0,C 180,E1 5281.617,E2 5281.617} C_VEL
LIN {X 0,Y 661.168,Z 1114.177,A -85,B 0,C 180,E1 5285.22,E2 5285.22} C_VEL
LIN {X 0,Y 659.28,Z 1144.051,A -85,B 0,C 180,E1 5289.189,E2 5289.189} C_VEL
LIN {X 0,Y 658.07,Z 1168.231,A -85,B 0,C 180,E1 5293.319,E2 5293.319} C_VEL
LIN {X 0,Y 657.465,Z 1185.217,A -85,B 0,C 180,E1 5297.093,E2 5297.093} C_VEL
LIN {X 0,Y 657.227,Z 1197.329,A -85,B 0,C 180,E1 5300.738,E2 5300.738} C_VEL
LIN {X 0,Y 657.103,Z 1205.909,A -85,B 0,C 180,E1 5304.721,E2 5304.721} C_VEL
LIN {X 0,Y 657.003,Z 1209.668,A -85,B 0,C 180,E1 5308.681,E2 5308.681} C_VEL
LIN {X 0,Y 657.204,Z 1208.945,A -85,B 0,C 180,E1 5312.635,E2 5312.635} C_VEL
LIN {X 0,Y 657.167,Z 1203.571,A -85,B 0,C 180,E1 5316.601,E2 5316.601} C_VEL
LIN {X 0,Y 657.379,Z 1192.318,A -85,B 0,C 180,E1 5320.931,E2 5320.931} C_VEL
LIN {X 0,Y 657.796,Z 1175.291,A -85,B 0,C 180,E1 5325.237,E2 5325.237} C_VEL
LIN {X 0,Y 658.607,Z 1155.299,A -85,B 0,C 180,E1 5329.028,E2 5329.028} C_VEL
LIN {X 0,Y 660.084,Z 1129.165,A -85,B 0,C 180,E1 5332.903,E2 5332.903} C_VEL
LIN {X 0,Y 662.404,Z 1096.461,A -85,B 0,C 180,E1 5336.778,E2 5336.778} C_VEL
LIN {X 0,Y 665.24,Z 1058.875,A -85,B 0,C 180,E1 5340.322,E2 5340.322} C_VEL
LIN {X 0,Y 668.48,Z 1019.131,A -85,B 0,C 180,E1 5343.33,E2 5343.33} C_VEL
LIN {X 0,Y 671.852,Z 975.716,A -85,B 0,C 180,E1 5345.93,E2 5345.93} C_VEL
LIN {X 0,Y 674.999,Z 931.384,A -85,B 0,C 180,E1 5347.978,E2 5347.978} C_VEL
LIN {X 0,Y 677.631,Z 883.522,A -85,B 0,C 180,E1 5349.595,E2 5349.595} C_VEL
LIN {X 0,Y 679.604,Z 835.939,A -85,B 0,C 180,E1 5350.648,E2 5350.648} C_VEL
LIN {X 0,Y 679.625,Z 804.505,A -85,B 0,C 180,E1 5351.129,E2 5351.129} C_VEL
LIN {X 0,Y 656.663,Z 763.269,A -85,B 0,C 180,E1 5353.509,E2 5353.509} C_VEL
LIN {X 0,Y 656.555,Z 762.06,A -85,B 0,C 180,E1 5353.571,E2 5353.571} C_VEL
LIN {X 0,Y 656.403,Z 762.06,A -85,B 0,C 180,E1 5358.113,E2 5358.113} C_VEL
LIN {X 0,Y 656.466,Z 762.06,A -85,B 0,C 180,E1 5363.673,E2 5363.673} C_VEL
LIN {X 0,Y 656.458,Z 762.06,A -85,B 0,C 180,E1 5368.397,E2 5368.397} C_VEL
LIN {X 0,Y 656.517,Z 762.06,A -85,B 0,C 180,E1 5374.062,E2 5374.062} C_VEL
LIN {X 0,Y 656.584,Z 762.06,A -85,B 0,C 180,E1 5379.799,E2 5379.799} C_VEL
LIN {X 0,Y 656.745,Z 762.06,A -85,B 0,C 180,E1 5385.099,E2 5385.099} C_VEL
LIN {X 0,Y 656.874,Z 762.06,A -85,B 0,C 180,E1 5390.727,E2 5390.727} C_VEL
LIN {X 0,Y 657.001,Z 762.06,A -85,B 0,C 180,E1 5396.036,E2 5396.036} C_VEL
LIN {X 0,Y 657.059,Z 762.06,A -85,B 0,C 180,E1 5399.992,E2 5399.992} C_VEL
LIN {X 0,Y 656.975,Z 762.06,A -85,B 0,C 180,E1 5405.271,E2 5405.271} C_VEL
LIN {X 0,Y 656.836,Z 762.06,A -85,B 0,C 180,E1 5410.596,E2 5410.596} C_VEL
LIN {X 0,Y 656.451,Z 762.06,A -85,B 0,C 180,E1 5416.025,E2 5416.025} C_VEL
LIN {X 0,Y 656.532,Z 762.06,A -85,B 0,C 180,E1 5421.598,E2 5421.598} C_VEL
LIN {X 0,Y 656.475,Z 762.06,A -85,B 0,C 180,E1 5426.141,E2 5426.141} C_VEL
LIN {X 0,Y 656.504,Z 762.06,A -85,B 0,C 180,E1 5431.61,E2 5431.61} C_VEL
LIN {X 0,Y 656.469,Z 762.06,A -85,B 0,C 180,E1 5436.747,E2 5436.747} C_VEL
LIN {X 0,Y 656.288,Z 762.06,A -85,B 0,C 180,E1 5442.541,E2 5442.541} C_VEL
LIN {X 0,Y 656.539,Z 762.858,A -85,B 0,C 180,E1 5446.871,E2 5446.871} C_VEL
LIN {X 0,Y 679.558,Z 804.599,A -85,B 0,C 180,E1 5449.28,E2 5449.28} C_VEL
LIN {X 0,Y 677.906,Z 850.929,A -85,B 0,C 180,E1 5450.298,E2 5450.298} C_VEL
LIN {X 0,Y 675.33,Z 895.079,A -85,B 0,C 180,E1 5451.732,E2 5451.732} C_VEL
LIN {X 0,Y 672.325,Z 940.408,A -85,B 0,C 180,E1 5453.745,E2 5453.745} C_VEL
LIN {X 0,Y 668.825,Z 984.166,A -85,B 0,C 180,E1 5456.294,E2 5456.294} C_VEL
LIN {X 0,Y 665.543,Z 1025.597,A -85,B 0,C 180,E1 5459.354,E2 5459.354} C_VEL
LIN {X 0,Y 662.387,Z 1065.145,A -85,B 0,C 180,E1 5463.038,E2 5463.038} C_VEL
LIN {X 0,Y 660.286,Z 1095.991,A -85,B 0,C 180,E1 5466.637,E2 5466.637} C_VEL
LIN {X 0,Y 658.748,Z 1121.818,A -85,B 0,C 180,E1 5470.362,E2 5470.362} C_VEL
LIN {X 0,Y 657.904,Z 1141.947,A -85,B 0,C 180,E1 5474.002,E2 5474.002} C_VEL
LIN {X 0,Y 657.338,Z 1159.047,A -85,B 0,C 180,E1 5478.06,E2 5478.06} C_VEL
LIN {X 0,Y 657.103,Z 1170.819,A -85,B 0,C 180,E1 5482.07,E2 5482.07} C_VEL
LIN {X 0,Y 657.013,Z 1177.732,A -85,B 0,C 180,E1 5486.044,E2 5486.044} C_VEL
LIN {X 0,Y 656.988,Z 1179.995,A -85,B 0,C 180,E1 5490.001,E2 5490.001} C_VEL
LIN {X 0,Y 657.113,Z 1177.625,A -85,B 0,C 180,E1 5493.957,E2 5493.957} C_VEL
LIN {X 0,Y 657.205,Z 1170.604,A -85,B 0,C 180,E1 5497.93,E2 5497.93} C_VEL
LIN {X 0,Y 657.525,Z 1157.439,A -85,B 0,C 180,E1 5502.295,E2 5502.295} C_VEL
LIN {X 0,Y 657.994,Z 1139.753,A -85,B 0,C 180,E1 5506.34,E2 5506.34} C_VEL
LIN {X 0,Y 659.136,Z 1116.001,A -85,B 0,C 180,E1 5510.465,E2 5510.465} C_VEL
LIN {X 0,Y 660.886,Z 1087.775,A -85,B 0,C 180,E1 5514.304,E2 5514.304} C_VEL
LIN {X 0,Y 663.371,Z 1053.747,A -85,B 0,C 180,E1 5518.023,E2 5518.023} C_VEL
LIN {X 0,Y 666.443,Z 1014.565,A -85,B 0,C 180,E1 5521.434,E2 5521.434} C_VEL
LIN {X 0,Y 669.699,Z 974.184,A -85,B 0,C 180,E1 5524.256,E2 5524.256} C_VEL
LIN {X 0,Y 673.004,Z 929.803,A -85,B 0,C 180,E1 5526.685,E2 5526.685} C_VEL
LIN {X 0,Y 676.04,Z 883.182,A -85,B 0,C 180,E1 5528.623,E2 5528.623} C_VEL
LIN {X 0,Y 678.443,Z 834.754,A -85,B 0,C 180,E1 5530.03,E2 5530.03} C_VEL
LIN {X 0,Y 679.208,Z 804.299,A -85,B 0,C 180,E1 5530.661,E2 5530.661} C_VEL
LIN {X 0,Y 656.677,Z 763.107,A -85,B 0,C 180,E1 5533.024,E2 5533.024} C_VEL
LIN {X 0,Y 656.59,Z 762.06,A -85,B 0,C 180,E1 5533.157,E2 5533.157} C_VEL
LIN {X 0,Y 656.343,Z 762.06,A -85,B 0,C 180,E1 5538.129,E2 5538.129} C_VEL
LIN {X 0,Y 656.449,Z 762.06,A -85,B 0,C 180,E1 5543.677,E2 5543.677} C_VEL
LIN {X 0,Y 656.421,Z 762.06,A -85,B 0,C 180,E1 5548.404,E2 5548.404} C_VEL
LIN {X 0,Y 656.433,Z 762.06,A -85,B 0,C 180,E1 5554.075,E2 5554.075} C_VEL
LIN {X 0,Y 656.457,Z 762.06,A -85,B 0,C 180,E1 5559.811,E2 5559.811} C_VEL
LIN {X 0,Y 656.591,Z 762.06,A -85,B 0,C 180,E1 5565.345,E2 5565.345} C_VEL
LIN {X 0,Y 656.863,Z 762.06,A -85,B 0,C 180,E1 5570.742,E2 5570.742} C_VEL
LIN {X 0,Y 657.024,Z 762.06,A -85,B 0,C 180,E1 5576.052,E2 5576.052} C_VEL
LIN {X 0,Y 657.164,Z 762.06,A -85,B 0,C 180,E1 5581.325,E2 5581.325} C_VEL
LIN {X 0,Y 656.844,Z 762.06,A -85,B 0,C 180,E1 5586.612,E2 5586.612} C_VEL
LIN {X 0,Y 656.796,Z 762.06,A -85,B 0,C 180,E1 5591.957,E2 5591.957} C_VEL
LIN {X 0,Y 656.837,Z 762.06,A -85,B 0,C 180,E1 5597.408,E2 5597.408} C_VEL
LIN {X 0,Y 656.671,Z 762.06,A -85,B 0,C 180,E1 5603.034,E2 5603.034} C_VEL
LIN {X 0,Y 656.614,Z 762.06,A -85,B 0,C 180,E1 5607.41,E2 5607.41} C_VEL
LIN {X 0,Y 656.553,Z 762.06,A -85,B 0,C 180,E1 5611.69,E2 5611.69} C_VEL
LIN {X 0,Y 652.535,Z 762.06,A -85,B 0,C 180,E1 5613.18,E2 5613.18} C_VEL
LIN {X 0,Y 648.536,Z 762.06,A -85,B 0,C 180,E1 5614.688,E2 5614.688} C_VEL
LIN {X 0,Y 648.457,Z 762.06,A -85,B 0,C 180,E1 5619.734,E2 5619.734} C_VEL
LIN {X 0,Y 648.643,Z 762.06,A -85,B 0,C 180,E1 5624.342,E2 5624.342} C_VEL
LIN {X 0,Y 648.616,Z 762.796,A -85,B 0,C 180,E1 5625.805,E2 5625.805} C_VEL
LIN {X 0,Y 657.493,Z 778.755,A -85,B 0,C 180,E1 5626.787,E2 5626.787} C_VEL
LIN {X 0,Y 674.107,Z 807.984,A -85,B 0,C 180,E1 5628.508,E2 5628.508} C_VEL
LIN {X 0,Y 672.784,Z 859.758,A -85,B 0,C 180,E1 5629.385,E2 5629.385} C_VEL
LIN {X 0,Y 670.188,Z 904.873,A -85,B 0,C 180,E1 5630.619,E2 5630.619} C_VEL
LIN {X 0,Y 667.084,Z 952.36,A -85,B 0,C 180,E1 5632.491,E2 5632.491} C_VEL
LIN {X 0,Y 663.291,Z 998.55,A -85,B 0,C 180,E1 5634.951,E2 5634.951} C_VEL
LIN {X 0,Y 659.795,Z 1039.86,A -85,B 0,C 180,E1 5637.771,E2 5637.771} C_VEL
LIN {X 0,Y 656.321,Z 1080.433,A -85,B 0,C 180,E1 5641.273,E2 5641.273} C_VEL
LIN {X 0,Y 653.647,Z 1113.67,A -85,B 0,C 180,E1 5644.852,E2 5644.852} C_VEL
LIN {X 0,Y 651.565,Z 1144.049,A -85,B 0,C 180,E1 5648.931,E2 5648.931} C_VEL
LIN {X 0,Y 650.289,Z 1168.233,A -85,B 0,C 180,E1 5653.113,E2 5653.113} C_VEL
LIN {X 0,Y 649.567,Z 1186.28,A -85,B 0,C 180,E1 5657.206,E2 5657.206} C_VEL
LIN {X 0,Y 649.271,Z 1199.109,A -85,B 0,C 180,E1 5661.301,E2 5661.301} C_VEL
LIN {X 0,Y 649.227,Z 1205.909,A -85,B 0,C 180,E1 5664.657,E2 5664.657} C_VEL
LIN {X 0,Y 649.128,Z 1209.668,A -85,B 0,C 180,E1 5668.665,E2 5668.665} C_VEL
LIN {X 0,Y 649.306,Z 1208.942,A -85,B 0,C 180,E1 5672.667,E2 5672.667} C_VEL
LIN {X 0,Y 649.271,Z 1203.571,A -85,B 0,C 180,E1 5676.682,E2 5676.682} C_VEL
LIN {X 0,Y 649.476,Z 1192.318,A -85,B 0,C 180,E1 5681.066,E2 5681.066} C_VEL
LIN {X 0,Y 649.969,Z 1175.293,A -85,B 0,C 180,E1 5685.425,E2 5685.425} C_VEL
LIN {X 0,Y 650.874,Z 1155.453,A -85,B 0,C 180,E1 5689.236,E2 5689.236} C_VEL
LIN {X 0,Y 652.482,Z 1129.163,A -85,B 0,C 180,E1 5693.185,E2 5693.185} C_VEL
LIN {X 0,Y 654.933,Z 1096.88,A -85,B 0,C 180,E1 5697.062,E2 5697.062} C_VEL
LIN {X 0,Y 658.114,Z 1058.874,A -85,B 0,C 180,E1 5700.685,E2 5700.685} C_VEL
LIN {X 0,Y 661.576,Z 1019.398,A -85,B 0,C 180,E1 5703.706,E2 5703.706} C_VEL
LIN {X 0,Y 665.299,Z 975.713,A -85,B 0,C 180,E1 5706.341,E2 5706.341} C_VEL
LIN {X 0,Y 668.632,Z 932.074,A -85,B 0,C 180,E1 5708.376,E2 5708.376} C_VEL
LIN {X 0,Y 671.449,Z 884.363,A -85,B 0,C 180,E1 5710.005,E2 5710.005} C_VEL
LIN {X 0,Y 673.531,Z 837.655,A -85,B 0,C 180,E1 5711.058,E2 5711.058} C_VEL
LIN {X 0,Y 673.565,Z 807.496,A -85,B 0,C 180,E1 5711.539,E2 5711.539} C_VEL
LIN {X 0,Y 648.807,Z 763.613,A -85,B 0,C 180,E1 5714.166,E2 5714.166} C_VEL
LIN {X 0,Y 648.644,Z 762.06,A -85,B 0,C 180,E1 5714.337,E2 5714.337} C_VEL
LIN {X 0,Y 648.507,Z 762.06,A -85,B 0,C 180,E1 5719.27,E2 5719.27} C_VEL
LIN {X 0,Y 648.513,Z 762.06,A -85,B 0,C 180,E1 5724.64,E2 5724.64} C_VEL
LIN {X 0,Y 648.539,Z 762.06,A -85,B 0,C 180,E1 5729.553,E2 5729.553} C_VEL
LIN {X 0,Y 648.631,Z 762.06,A -85,B 0,C 180,E1 5735.308,E2 5735.308} C_VEL
LIN {X 0,Y 648.693,Z 762.06,A -85,B 0,C 180,E1 5740.961,E2 5740.961} C_VEL
LIN {X 0,Y 648.853,Z 762.06,A -85,B 0,C 180,E1 5745.15,E2 5745.15} C_VEL
LIN {X 0,Y 648.955,Z 762.06,A -85,B 0,C 180,E1 5750.612,E2 5750.612} C_VEL
LIN {X 0,Y 649.119,Z 762.06,A -85,B 0,C 180,E1 5755.988,E2 5755.988} C_VEL
LIN {X 0,Y 649.172,Z 762.06,A -85,B 0,C 180,E1 5759.992,E2 5759.992} C_VEL
LIN {X 0,Y 649.067,Z 762.06,A -85,B 0,C 180,E1 5765.335,E2 5765.335} C_VEL
LIN {X 0,Y 648.911,Z 762.06,A -85,B 0,C 180,E1 5770.727,E2 5770.727} C_VEL
LIN {X 0,Y 648.517,Z 762.06,A -85,B 0,C 180,E1 5776.227,E2 5776.227} C_VEL
LIN {X 0,Y 648.605,Z 762.06,A -85,B 0,C 180,E1 5781.875,E2 5781.875} C_VEL
LIN {X 0,Y 648.576,Z 762.06,A -85,B 0,C 180,E1 5786.263,E2 5786.263} C_VEL
LIN {X 0,Y 648.555,Z 762.06,A -85,B 0,C 180,E1 5790.823,E2 5790.823} C_VEL
LIN {X 0,Y 648.555,Z 762.06,A -85,B 0,C 180,E1 5795.611,E2 5795.611} C_VEL
LIN {X 0,Y 648.392,Z 762.06,A -85,B 0,C 180,E1 5800.718,E2 5800.718} C_VEL
LIN {X 0,Y 648.484,Z 762.173,A -85,B 0,C 180,E1 5806.192,E2 5806.192} C_VEL
LIN {X 0,Y 650.857,Z 767.672,A -85,B 0,C 180,E1 5806.473,E2 5806.473} C_VEL
LIN {X 0,Y 673.506,Z 807.673,A -85,B 0,C 180,E1 5808.895,E2 5808.895} C_VEL
LIN {X 0,Y 671.581,Z 854.262,A -85,B 0,C 180,E1 5809.956,E2 5809.956} C_VEL
LIN {X 0,Y 668.913,Z 896.709,A -85,B 0,C 180,E1 5811.367,E2 5811.367} C_VEL
LIN {X 0,Y 665.726,Z 941.067,A -85,B 0,C 180,E1 5813.366,E2 5813.366} C_VEL
LIN {X 0,Y 661.889,Z 985.53,A -85,B 0,C 180,E1 5815.991,E2 5815.991} C_VEL
LIN {X 0,Y 658.382,Z 1025.833,A -85,B 0,C 180,E1 5819.006,E2 5819.006} C_VEL
LIN {X 0,Y 655.023,Z 1065.27,A -85,B 0,C 180,E1 5822.724,E2 5822.724} C_VEL
LIN {X 0,Y 652.661,Z 1096.441,A -85,B 0,C 180,E1 5826.409,E2 5826.409} C_VEL
LIN {X 0,Y 651.016,Z 1122.316,A -85,B 0,C 180,E1 5830.201,E2 5830.201} C_VEL
LIN {X 0,Y 649.987,Z 1143.667,A -85,B 0,C 180,E1 5834.169,E2 5834.169} C_VEL
LIN {X 0,Y 649.443,Z 1160.203,A -85,B 0,C 180,E1 5838.254,E2 5838.254} C_VEL
LIN {X 0,Y 649.239,Z 1170.815,A -85,B 0,C 180,E1 5841.973,E2 5841.973} C_VEL
LIN {X 0,Y 649.113,Z 1177.731,A -85,B 0,C 180,E1 5845.996,E2 5845.996} C_VEL
LIN {X 0,Y 649.105,Z 1179.995,A -85,B 0,C 180,E1 5850.001,E2 5850.001} C_VEL
LIN {X 0,Y 649.238,Z 1177.626,A -85,B 0,C 180,E1 5854.005,E2 5854.005} C_VEL
LIN {X 0,Y 649.352,Z 1170.603,A -85,B 0,C 180,E1 5858.027,E2 5858.027} C_VEL
LIN {X 0,Y 649.647,Z 1157.618,A -85,B 0,C 180,E1 5862.397,E2 5862.397} C_VEL
LIN {X 0,Y 650.201,Z 1139.754,A -85,B 0,C 180,E1 5866.542,E2 5866.542} C_VEL
LIN {X 0,Y 651.473,Z 1116.007,A -85,B 0,C 180,E1 5870.716,E2 5870.716} C_VEL
LIN {X 0,Y 653.331,Z 1087.777,A -85,B 0,C 180,E1 5874.604,E2 5874.604} C_VEL
LIN {X 0,Y 656.045,Z 1053.749,A -85,B 0,C 180,E1 5878.365,E2 5878.365} C_VEL
LIN {X 0,Y 659.381,Z 1014.571,A -85,B 0,C 180,E1 5881.81,E2 5881.81} C_VEL
LIN {X 0,Y 662.95,Z 974.013,A -85,B 0,C 180,E1 5884.666,E2 5884.666} C_VEL
LIN {X 0,Y 666.498,Z 929.945,A -85,B 0,C 180,E1 5887.096,E2 5887.096} C_VEL
LIN {X 0,Y 669.706,Z 884.603,A -85,B 0,C 180,E1 5889.004,E2 5889.004} C_VEL
LIN {X 0,Y 672.383,Z 834.673,A -85,B 0,C 180,E1 5890.467,E2 5890.467} C_VEL
LIN {X 0,Y 673.213,Z 807.549,A -85,B 0,C 180,E1 5891.039,E2 5891.039} C_VEL
LIN {X 0,Y 648.72,Z 763.084,A -85,B 0,C 180,E1 5893.685,E2 5893.685} C_VEL
LIN {X 0,Y 648.655,Z 762.06,A -85,B 0,C 180,E1 5893.784,E2 5893.784} C_VEL
LIN {X 0,Y 648.471,Z 762.06,A -85,B 0,C 180,E1 5899.288,E2 5899.288} C_VEL
LIN {X 0,Y 648.517,Z 762.06,A -85,B 0,C 180,E1 5904.641,E2 5904.641} C_VEL
LIN {X 0,Y 648.489,Z 762.06,A -85,B 0,C 180,E1 5909.563,E2 5909.563} C_VEL
LIN {X 0,Y 648.516,Z 762.06,A -85,B 0,C 180,E1 5915.214,E2 5915.214} C_VEL
LIN {X 0,Y 648.526,Z 762.06,A -85,B 0,C 180,E1 5919.554,E2 5919.554} C_VEL
LIN {X 0,Y 648.695,Z 762.06,A -85,B 0,C 180,E1 5925.163,E2 5925.163} C_VEL
LIN {X 0,Y 648.948,Z 762.06,A -85,B 0,C 180,E1 5930.628,E2 5930.628} C_VEL
LIN {X 0,Y 649.135,Z 762.06,A -85,B 0,C 180,E1 5936.004,E2 5936.004} C_VEL
LIN {X 0,Y 649.272,Z 762.06,A -85,B 0,C 180,E1 5941.341,E2 5941.341} C_VEL
LIN {X 0,Y 648.959,Z 762.06,A -85,B 0,C 180,E1 5946.693,E2 5946.693} C_VEL
LIN {X 0,Y 648.888,Z 762.06,A -85,B 0,C 180,E1 5952.105,E2 5952.105} C_VEL
LIN {X 0,Y 648.904,Z 762.06,A -85,B 0,C 180,E1 5957.628,E2 5957.628} C_VEL
LIN {X 0,Y 648.787,Z 762.06,A -85,B 0,C 180,E1 5961.885,E2 5961.885} C_VEL
LIN {X 0,Y 648.709,Z 762.06,A -85,B 0,C 180,E1 5966.274,E2 5966.274} C_VEL
LIN {X 0,Y 648.547,Z 762.06,A -85,B 0,C 180,E1 5971.688,E2 5971.688} C_VEL
LIN {X 0,Y 648.536,Z 762.06,A -85,B 0,C 180,E1 5974.688,E2 5974.688} C_VEL
LIN {X 0,Y 647.254,Z 762.06,A -85,B 0,C 180,E1 5975.454,E2 5975.454} C_VEL
LIN {X 0,Y 640.624,Z 762.06,A -85,B 0,C 180,E1 5977.535,E2 5977.535} C_VEL
LIN {X 0,Y 640.548,Z 762.06,A -85,B 0,C 180,E1 5977.732,E2 5977.732} C_VEL
LIN {X 0,Y 640.71,Z 762.06,A -85,B 0,C 180,E1 5983.158,E2 5983.158} C_VEL
LIN {X 0,Y 640.731,Z 762.849,A -85,B 0,C 180,E1 5985.118,E2 5985.118} C_VEL
LIN {X 0,Y 649.717,Z 778.822,A -85,B 0,C 180,E1 5986.141,E2 5986.141} C_VEL
LIN {X 0,Y 668.126,Z 811.117,A -85,B 0,C 180,E1 5988.097,E2 5988.097} C_VEL
LIN {X 0,Y 666.595,Z 862.335,A -85,B 0,C 180,E1 5988.998,E2 5988.998} C_VEL
LIN {X 0,Y 663.831,Z 907.357,A -85,B 0,C 180,E1 5990.261,E2 5990.261} C_VEL
LIN {X 0,Y 660.557,Z 953.762,A -85,B 0,C 180,E1 5992.131,E2 5992.131} C_VEL
LIN {X 0,Y 656.501,Z 999.747,A -85,B 0,C 180,E1 5994.614,E2 5994.614} C_VEL
LIN {X 0,Y 652.746,Z 1040.594,A -85,B 0,C 180,E1 5997.443,E2 5997.443} C_VEL
LIN {X 0,Y 648.95,Z 1081.701,A -85,B 0,C 180,E1 6001.042,E2 6001.042} C_VEL
LIN {X 0,Y 645.978,Z 1116.178,A -85,B 0,C 180,E1 6004.849,E2 6004.849} C_VEL
LIN {X 0,Y 643.829,Z 1145.187,A -85,B 0,C 180,E1 6008.846,E2 6008.846} C_VEL
LIN {X 0,Y 642.409,Z 1169.977,A -85,B 0,C 180,E1 6013.252,E2 6013.252} C_VEL
LIN {X 0,Y 641.711,Z 1186.38,A -85,B 0,C 180,E1 6017.072,E2 6017.072} C_VEL
LIN {X 0,Y 641.399,Z 1199.267,A -85,B 0,C 180,E1 6021.259,E2 6021.259} C_VEL
LIN {X 0,Y 641.329,Z 1205.909,A -85,B 0,C 180,E1 6024.591,E2 6024.591} C_VEL
LIN {X 0,Y 641.228,Z 1209.668,A -85,B 0,C 180,E1 6028.649,E2 6028.649} C_VEL
LIN {X 0,Y 641.399,Z 1208.939,A -85,B 0,C 180,E1 6032.7,E2 6032.7} C_VEL
LIN {X 0,Y 641.37,Z 1203.571,A -85,B 0,C 180,E1 6036.765,E2 6036.765} C_VEL
LIN {X 0,Y 641.577,Z 1192.317,A -85,B 0,C 180,E1 6041.204,E2 6041.204} C_VEL
LIN {X 0,Y 642.109,Z 1176.264,A -85,B 0,C 180,E1 6045.399,E2 6045.399} C_VEL
LIN {X 0,Y 643.143,Z 1155.818,A -85,B 0,C 180,E1 6049.41,E2 6049.41} C_VEL
LIN {X 0,Y 644.897,Z 1129.161,A -85,B 0,C 180,E1 6053.474,E2 6053.474} C_VEL
LIN {X 0,Y 647.596,Z 1096.664,A -85,B 0,C 180,E1 6057.419,E2 6057.419} C_VEL
LIN {X 0,Y 651.012,Z 1058.892,A -85,B 0,C 180,E1 6061.055,E2 6061.055} C_VEL
LIN {X 0,Y 654.653,Z 1020.414,A -85,B 0,C 180,E1 6064.037,E2 6064.037} C_VEL
LIN {X 0,Y 658.637,Z 976.89,A -85,B 0,C 180,E1 6066.697,E2 6066.697} C_VEL
LIN {X 0,Y 662.267,Z 933.056,A -85,B 0,C 180,E1 6068.771,E2 6068.771} C_VEL
LIN {X 0,Y 665.214,Z 886.297,A -85,B 0,C 180,E1 6070.393,E2 6070.393} C_VEL
LIN {X 0,Y 667.521,Z 838.746,A -85,B 0,C 180,E1 6071.486,E2 6071.486} C_VEL
LIN {X 0,Y 667.788,Z 810.962,A -85,B 0,C 180,E1 6071.931,E2 6071.931} C_VEL
LIN {X 0,Y 642.836,Z 767.456,A -85,B 0,C 180,E1 6074.626,E2 6074.626} C_VEL
LIN {X 0,Y 640.683,Z 762.06,A -85,B 0,C 180,E1 6074.958,E2 6074.958} C_VEL
LIN {X 0,Y 640.579,Z 762.06,A -85,B 0,C 180,E1 6080.433,E2 6080.433} C_VEL
LIN {X 0,Y 640.597,Z 762.06,A -85,B 0,C 180,E1 6085.65,E2 6085.65} C_VEL
LIN {X 0,Y 640.62,Z 762.06,A -85,B 0,C 180,E1 6090.78,E2 6090.78} C_VEL
LIN {X 0,Y 640.684,Z 762.06,A -85,B 0,C 180,E1 6094.873,E2 6094.873} C_VEL
LIN {X 0,Y 640.757,Z 762.06,A -85,B 0,C 180,E1 6100.715,E2 6100.715} C_VEL
LIN {X 0,Y 640.974,Z 762.06,A -85,B 0,C 180,E1 6105.144,E2 6105.144} C_VEL
LIN {X 0,Y 641.039,Z 762.06,A -85,B 0,C 180,E1 6110.495,E2 6110.495} C_VEL
LIN {X 0,Y 641.213,Z 762.06,A -85,B 0,C 180,E1 6115.939,E2 6115.939} C_VEL
LIN {X 0,Y 641.272,Z 762.06,A -85,B 0,C 180,E1 6119.992,E2 6119.992} C_VEL
LIN {X 0,Y 641.227,Z 762.06,A -85,B 0,C 180,E1 6124.046,E2 6124.046} C_VEL
LIN {X 0,Y 641.019,Z 762.06,A -85,B 0,C 180,E1 6129.489,E2 6129.489} C_VEL
LIN {X 0,Y 640.744,Z 762.06,A -85,B 0,C 180,E1 6135.026,E2 6135.026} C_VEL
LIN {X 0,Y 640.689,Z 762.06,A -85,B 0,C 180,E1 6140.708,E2 6140.708} C_VEL
LIN {X 0,Y 640.668,Z 762.06,A -85,B 0,C 180,E1 6146.327,E2 6146.327} C_VEL
LIN {X 0,Y 640.583,Z 762.06,A -85,B 0,C 180,E1 6151.874,E2 6151.874} C_VEL
LIN {X 0,Y 640.552,Z 762.06,A -85,B 0,C 180,E1 6156.671,E2 6156.671} C_VEL
LIN {X 0,Y 640.48,Z 762.06,A -85,B 0,C 180,E1 6161.33,E2 6161.33} C_VEL
LIN {X 0,Y 640.568,Z 762.315,A -85,B 0,C 180,E1 6165.512,E2 6165.512} C_VEL
LIN {X 0,Y 643.247,Z 767.982,A -85,B 0,C 180,E1 6165.832,E2 6165.832} C_VEL
LIN {X 0,Y 667.419,Z 810.887,A -85,B 0,C 180,E1 6168.508,E2 6168.508} C_VEL
LIN {X 0,Y 665.292,Z 857.884,A -85,B 0,C 180,E1 6169.619,E2 6169.619} C_VEL
LIN {X 0,Y 662.453,Z 899.349,A -85,B 0,C 180,E1 6171.035,E2 6171.035} C_VEL
LIN {X 0,Y 659.079,Z 942.358,A -85,B 0,C 180,E1 6173.014,E2 6173.014} C_VEL
LIN {X 0,Y 654.946,Z 986.909,A -85,B 0,C 180,E1 6175.681,E2 6175.681} C_VEL
LIN {X 0,Y 651.177,Z 1027.073,A -85,B 0,C 180,E1 6178.74,E2 6178.74} C_VEL
LIN {X 0,Y 647.677,Z 1065.527,A -85,B 0,C 180,E1 6182.417,E2 6182.417} C_VEL
LIN {X 0,Y 645.028,Z 1097.295,A -85,B 0,C 180,E1 6186.229,E2 6186.229} C_VEL
LIN {X 0,Y 643.286,Z 1122.855,A -85,B 0,C 180,E1 6190.043,E2 6190.043} C_VEL
LIN {X 0,Y 642.227,Z 1143.411,A -85,B 0,C 180,E1 6193.914,E2 6193.914} C_VEL
LIN {X 0,Y 641.584,Z 1160.198,A -85,B 0,C 180,E1 6198.108,E2 6198.108} C_VEL
LIN {X 0,Y 641.343,Z 1170.81,A -85,B 0,C 180,E1 6201.874,E2 6201.874} C_VEL
LIN {X 0,Y 641.21,Z 1177.731,A -85,B 0,C 180,E1 6205.947,E2 6205.947} C_VEL
LIN {X 0,Y 641.205,Z 1179.996,A -85,B 0,C 180,E1 6210.001,E2 6210.001} C_VEL
LIN {X 0,Y 641.336,Z 1177.626,A -85,B 0,C 180,E1 6214.054,E2 6214.054} C_VEL
LIN {X 0,Y 641.526,Z 1169.769,A -85,B 0,C 180,E1 6218.488,E2 6218.488} C_VEL
LIN {X 0,Y 641.756,Z 1157.62,A -85,B 0,C 180,E1 6222.552,E2 6222.552} C_VEL
LIN {X 0,Y 642.396,Z 1139.756,A -85,B 0,C 180,E1 6226.748,E2 6226.748} C_VEL
LIN {X 0,Y 643.811,Z 1116.012,A -85,B 0,C 180,E1 6230.974,E2 6230.974} C_VEL
LIN {X 0,Y 645.835,Z 1087.78,A -85,B 0,C 180,E1 6234.909,E2 6234.909} C_VEL
LIN {X 0,Y 648.726,Z 1053.849,A -85,B 0,C 180,E1 6238.704,E2 6238.704} C_VEL
LIN {X 0,Y 652.363,Z 1014.577,A -85,B 0,C 180,E1 6242.193,E2 6242.193} C_VEL
LIN {X 0,Y 656.212,Z 974.413,A -85,B 0,C 180,E1 6245.048,E2 6245.048} C_VEL
LIN {X 0,Y 659.916,Z 931.406,A -85,B 0,C 180,E1 6247.45,E2 6247.45} C_VEL
LIN {X 0,Y 663.432,Z 885.454,A -85,B 0,C 180,E1 6249.409,E2 6249.409} C_VEL
LIN {X 0,Y 666.23,Z 836.814,A -85,B 0,C 180,E1 6250.862,E2 6250.862} C_VEL
LIN {X 0,Y 667.008,Z 810.603,A -85,B 0,C 180,E1 6251.439,E2 6251.439} C_VEL
LIN {X 0,Y 642.913,Z 767.505,A -85,B 0,C 180,E1 6254.114,E2 6254.114} C_VEL
LIN {X 0,Y 640.711,Z 762.06,A -85,B 0,C 180,E1 6254.491,E2 6254.491} C_VEL
LIN {X 0,Y 640.554,Z 762.06,A -85,B 0,C 180,E1 6260.452,E2 6260.452} C_VEL
LIN {X 0,Y 640.555,Z 762.06,A -85,B 0,C 180,E1 6265.658,E2 6265.658} C_VEL
LIN {X 0,Y 640.57,Z 762.06,A -85,B 0,C 180,E1 6270.791,E2 6270.791} C_VEL
LIN {X 0,Y 640.579,Z 762.06,A -85,B 0,C 180,E1 6274.886,E2 6274.886} C_VEL
LIN {X 0,Y 640.617,Z 762.06,A -85,B 0,C 180,E1 6279.29,E2 6279.29} C_VEL
LIN {X 0,Y 640.801,Z 762.06,A -85,B 0,C 180,E1 6285.207,E2 6285.207} C_VEL
LIN {X 0,Y 641.035,Z 762.06,A -85,B 0,C 180,E1 6290.511,E2 6290.511} C_VEL
LIN {X 0,Y 641.223,Z 762.06,A -85,B 0,C 180,E1 6295.954,E2 6295.954} C_VEL
LIN {X 0,Y 641.366,Z 762.06,A -85,B 0,C 180,E1 6301.358,E2 6301.358} C_VEL
LIN {X 0,Y 641.05,Z 762.06,A -85,B 0,C 180,E1 6306.776,E2 6306.776} C_VEL
LIN {X 0,Y 640.968,Z 762.06,A -85,B 0,C 180,E1 6312.257,E2 6312.257} C_VEL
LIN {X 0,Y 640.972,Z 762.06,A -85,B 0,C 180,E1 6317.853,E2 6317.853} C_VEL
LIN {X 0,Y 640.82,Z 762.06,A -85,B 0,C 180,E1 6323.123,E2 6323.123} C_VEL
LIN {X 0,Y 640.722,Z 762.06,A -85,B 0,C 180,E1 6328.149,E2 6328.149} C_VEL
LIN {X 0,Y 640.684,Z 762.06,A -85,B 0,C 180,E1 6332.857,E2 6332.857} C_VEL
LIN {X 0,Y 640.548,Z 762.06,A -85,B 0,C 180,E1 6337.732,E2 6337.732} C_VEL
LIN {X 0,Y 638.071,Z 762.06,A -85,B 0,C 180,E1 6338.877,E2 6338.877} C_VEL
LIN {X 0,Y 632.693,Z 762.06,A -85,B 0,C 180,E1 6340.587,E2 6340.587} C_VEL
LIN {X 0,Y 632.595,Z 762.06,A -85,B 0,C 180,E1 6340.784,E2 6340.784} C_VEL
LIN {X 0,Y 632.734,Z 762.06,A -85,B 0,C 180,E1 6344.373,E2 6344.373} C_VEL
LIN {X 0,Y 635.253,Z 767.82,A -85,B 0,C 180,E1 6344.706,E2 6344.706} C_VEL
LIN {X 0,Y 662.271,Z 814.308,A -85,B 0,C 180,E1 6347.687,E2 6347.687} C_VEL
LIN {X 0,Y 660.462,Z 865.075,A -85,B 0,C 180,E1 6348.61,E2 6348.61} C_VEL
LIN {X 0,Y 657.46,Z 911.07,A -85,B 0,C 180,E1 6349.942,E2 6349.942} C_VEL
LIN {X 0,Y 653.806,Z 957.081,A -85,B 0,C 180,E1 6351.854,E2 6351.854} C_VEL
LIN {X 0,Y 649.465,Z 1003.575,A -85,B 0,C 180,E1 6354.431,E2 6354.431} C_VEL
LIN {X 0,Y 645.36,Z 1045.103,A -85,B 0,C 180,E1 6357.415,E2 6357.415} C_VEL
LIN {X 0,Y 641.509,Z 1083.947,A -85,B 0,C 180,E1 6360.907,E2 6360.907} C_VEL
LIN {X 0,Y 638.341,Z 1118.133,A -85,B 0,C 180,E1 6364.779,E2 6364.779} C_VEL
LIN {X 0,Y 636.06,Z 1146.456,A -85,B 0,C 180,E1 6368.786,E2 6368.786} C_VEL
LIN {X 0,Y 634.613,Z 1170.211,A -85,B 0,C 180,E1 6373.088,E2 6373.088} C_VEL
LIN {X 0,Y 633.808,Z 1187.677,A -85,B 0,C 180,E1 6377.259,E2 6377.259} C_VEL
LIN {X 0,Y 633.517,Z 1199.102,A -85,B 0,C 180,E1 6381.08,E2 6381.08} C_VEL
LIN {X 0,Y 633.43,Z 1205.909,A -85,B 0,C 180,E1 6384.524,E2 6384.524} C_VEL
LIN {X 0,Y 633.349,Z 1209.667,A -85,B 0,C 180,E1 6388.632,E2 6388.632} C_VEL
LIN {X 0,Y 633.509,Z 1208.936,A -85,B 0,C 180,E1 6392.734,E2 6392.734} C_VEL
LIN {X 0,Y 633.471,Z 1203.572,A -85,B 0,C 180,E1 6396.849,E2 6396.849} C_VEL
LIN {X 0,Y 633.696,Z 1193.421,A -85,B 0,C 180,E1 6400.997,E2 6400.997} C_VEL
LIN {X 0,Y 634.264,Z 1177.053,A -85,B 0,C 180,E1 6405.414,E2 6405.414} C_VEL
LIN {X 0,Y 635.4,Z 1155.963,A -85,B 0,C 180,E1 6409.63,E2 6409.63} C_VEL
LIN {X 0,Y 637.228,Z 1130.482,A -85,B 0,C 180,E1 6413.588,E2 6413.588} C_VEL
LIN {X 0,Y 640.119,Z 1097.859,A -85,B 0,C 180,E1 6417.626,E2 6417.626} C_VEL
LIN {X 0,Y 643.664,Z 1061.657,A -85,B 0,C 180,E1 6421.19,E2 6421.19} C_VEL
LIN {X 0,Y 647.713,Z 1022.084,A -85,B 0,C 180,E1 6424.33,E2 6424.33} C_VEL
LIN {X 0,Y 651.839,Z 979.732,A -85,B 0,C 180,E1 6426.97,E2 6426.97} C_VEL
LIN {X 0,Y 655.713,Z 935.988,A -85,B 0,C 180,E1 6429.09,E2 6429.09} C_VEL
LIN {X 0,Y 658.927,Z 889.846,A -85,B 0,C 180,E1 6430.742,E2 6430.742} C_VEL
LIN {X 0,Y 661.513,Z 840.673,A -85,B 0,C 180,E1 6431.904,E2 6431.904} C_VEL
LIN {X 0,Y 661.776,Z 813.84,A -85,B 0,C 180,E1 6432.359,E2 6432.359} C_VEL
LIN {X 0,Y 637.74,Z 772.197,A -85,B 0,C 180,E1 6435.003,E2 6435.003} C_VEL
LIN {X 0,Y 632.806,Z 763.189,A -85,B 0,C 180,E1 6435.59,E2 6435.59} C_VEL
LIN {X 0,Y 632.695,Z 762.06,A -85,B 0,C 180,E1 6435.766,E2 6435.766} C_VEL
LIN {X 0,Y 632.665,Z 762.06,A -85,B 0,C 180,E1 6441.606,E2 6441.606} C_VEL
LIN {X 0,Y 632.666,Z 762.06,A -85,B 0,C 180,E1 6446.716,E2 6446.716} C_VEL
LIN {X 0,Y 632.677,Z 762.06,A -85,B 0,C 180,E1 6452.093,E2 6452.093} C_VEL
LIN {X 0,Y 632.758,Z 762.06,A -85,B 0,C 180,E1 6457.531,E2 6457.531} C_VEL
LIN {X 0,Y 632.997,Z 762.06,A -85,B 0,C 180,E1 6463.347,E2 6463.347} C_VEL
LIN {X 0,Y 633.077,Z 762.06,A -85,B 0,C 180,E1 6468.985,E2 6468.985} C_VEL
LIN {X 0,Y 633.275,Z 762.06,A -85,B 0,C 180,E1 6474.516,E2 6474.516} C_VEL
LIN {X 0,Y 633.399,Z 762.06,A -85,B 0,C 180,E1 6479.992,E2 6479.992} C_VEL
LIN {X 0,Y 633.327,Z 762.06,A -85,B 0,C 180,E1 6484.096,E2 6484.096} C_VEL
LIN {X 0,Y 633.104,Z 762.06,A -85,B 0,C 180,E1 6489.609,E2 6489.609} C_VEL
LIN {X 0,Y 632.865,Z 762.06,A -85,B 0,C 180,E1 6493.804,E2 6493.804} C_VEL
LIN {X 0,Y 632.744,Z 762.06,A -85,B 0,C 180,E1 6499.522,E2 6499.522} C_VEL
LIN {X 0,Y 632.768,Z 762.06,A -85,B 0,C 180,E1 6504.843,E2 6504.843} C_VEL
LIN {X 0,Y 632.687,Z 762.06,A -85,B 0,C 180,E1 6510.705,E2 6510.705} C_VEL
LIN {X 0,Y 632.643,Z 762.06,A -85,B 0,C 180,E1 6515.698,E2 6515.698} C_VEL
LIN {X 0,Y 632.548,Z 762.06,A -85,B 0,C 180,E1 6520.15,E2 6520.15} C_VEL
LIN {X 0,Y 632.585,Z 762.06,A -85,B 0,C 180,E1 6524.772,E2 6524.772} C_VEL
LIN {X 0,Y 635.082,Z 767.786,A -85,B 0,C 180,E1 6525.106,E2 6525.106} C_VEL
LIN {X 0,Y 660.156,Z 811.54,A -85,B 0,C 180,E1 6527.965,E2 6527.965} C_VEL
LIN {X 0,Y 661.232,Z 817.016,A -85,B 0,C 180,E1 6528.171,E2 6528.171} C_VEL
LIN {X 0,Y 658.699,Z 865.929,A -85,B 0,C 180,E1 6529.404,E2 6529.404} C_VEL
LIN {X 0,Y 655.473,Z 908.317,A -85,B 0,C 180,E1 6530.964,E2 6530.964} C_VEL
LIN {X 0,Y 651.572,Z 952.653,A -85,B 0,C 180,E1 6533.146,E2 6533.146} C_VEL
LIN {X 0,Y 647.636,Z 993.063,A -85,B 0,C 180,E1 6535.696,E2 6535.696} C_VEL
LIN {X 0,Y 643.406,Z 1034.155,A -85,B 0,C 180,E1 6538.985,E2 6538.985} C_VEL
LIN {X 0,Y 639.949,Z 1069.222,A -85,B 0,C 180,E1 6542.482,E2 6542.482} C_VEL
LIN {X 0,Y 637.132,Z 1102.127,A -85,B 0,C 180,E1 6546.593,E2 6546.593} C_VEL
LIN {X 0,Y 635.278,Z 1127.209,A -85,B 0,C 180,E1 6550.549,E2 6550.549} C_VEL
LIN {X 0,Y 634.178,Z 1148.208,A -85,B 0,C 180,E1 6554.806,E2 6554.806} C_VEL
LIN {X 0,Y 633.636,Z 1163.552,A -85,B 0,C 180,E1 6559.002,E2 6559.002} C_VEL
LIN {X 0,Y 633.501,Z 1173.656,A -85,B 0,C 180,E1 6563.151,E2 6563.151} C_VEL
LIN {X 0,Y 633.354,Z 1178.97,A -85,B 0,C 180,E1 6567.266,E2 6567.266} C_VEL
LIN {X 0,Y 633.426,Z 1179.656,A -85,B 0,C 180,E1 6571.368,E2 6571.368} C_VEL
LIN {X 0,Y 633.506,Z 1175.842,A -85,B 0,C 180,E1 6575.476,E2 6575.476} C_VEL
LIN {X 0,Y 633.549,Z 1167.209,A -85,B 0,C 180,E1 6579.612,E2 6579.612} C_VEL
LIN {X 0,Y 633.981,Z 1153.53,A -85,B 0,C 180,E1 6583.79,E2 6583.79} C_VEL
LIN {X 0,Y 634.855,Z 1134.499,A -85,B 0,C 180,E1 6588.026,E2 6588.026} C_VEL
LIN {X 0,Y 636.483,Z 1110.232,A -85,B 0,C 180,E1 6592.13,E2 6592.13} C_VEL
LIN {X 0,Y 638.953,Z 1080.7,A -85,B 0,C 180,E1 6596.103,E2 6596.103} C_VEL
LIN {X 0,Y 642.213,Z 1046.253,A -85,B 0,C 180,E1 6599.797,E2 6599.797} C_VEL
LIN {X 0,Y 646.093,Z 1007.87,A -85,B 0,C 180,E1 6603.121,E2 6603.121} C_VEL
LIN {X 0,Y 650.426,Z 964.013,A -85,B 0,C 180,E1 6606.107,E2 6606.107} C_VEL
LIN {X 0,Y 654.481,Z 921.653,A -85,B 0,C 180,E1 6608.352,E2 6608.352} C_VEL
LIN {X 0,Y 657.839,Z 877.775,A -85,B 0,C 180,E1 6610.113,E2 6610.113} C_VEL
LIN {X 0,Y 660.464,Z 833.226,A -85,B 0,C 180,E1 6611.396,E2 6611.396} C_VEL
LIN {X 0,Y 660.909,Z 813.679,A -85,B 0,C 180,E1 6611.839,E2 6611.839} C_VEL
LIN {X 0,Y 638.156,Z 772.729,A -85,B 0,C 180,E1 6614.451,E2 6614.451} C_VEL
LIN {X 0,Y 632.816,Z 763.013,A -85,B 0,C 180,E1 6615.085,E2 6615.085} C_VEL
LIN {X 0,Y 632.744,Z 762.06,A -85,B 0,C 180,E1 6615.267,E2 6615.267} C_VEL
LIN {X 0,Y 632.623,Z 762.06,A -85,B 0,C 180,E1 6619.856,E2 6619.856} C_VEL
LIN {X 0,Y 632.61,Z 762.06,A -85,B 0,C 180,E1 6625.035,E2 6625.035} C_VEL
LIN {X 0,Y 632.607,Z 762.06,A -85,B 0,C 180,E1 6629.906,E2 6629.906} C_VEL
LIN {X 0,Y 632.643,Z 762.06,A -85,B 0,C 180,E1 6635.185,E2 6635.185} C_VEL
LIN {X 0,Y 632.689,Z 762.06,A -85,B 0,C 180,E1 6640.476,E2 6640.476} C_VEL
LIN {X 0,Y 632.881,Z 762.06,A -85,B 0,C 180,E1 6646.196,E2 6646.196} C_VEL
LIN {X 0,Y 633.239,Z 762.06,A -85,B 0,C 180,E1 6651.777,E2 6651.777} C_VEL
LIN {X 0,Y 633.43,Z 762.06,A -85,B 0,C 180,E1 6657.274,E2 6657.274} C_VEL
LIN {X 0,Y 633.273,Z 762.06,A -85,B 0,C 180,E1 6662.743,E2 6662.743} C_VEL
LIN {X 0,Y 633.173,Z 762.06,A -85,B 0,C 180,E1 6668.24,E2 6668.24} C_VEL
LIN {X 0,Y 633.065,Z 762.06,A -85,B 0,C 180,E1 6673.816,E2 6673.816} C_VEL
LIN {X 0,Y 633.058,Z 762.06,A -85,B 0,C 180,E1 6678.084,E2 6678.084} C_VEL
LIN {X 0,Y 632.919,Z 762.06,A -85,B 0,C 180,E1 6682.463,E2 6682.463} C_VEL
LIN {X 0,Y 632.804,Z 762.06,A -85,B 0,C 180,E1 6687.926,E2 6687.926} C_VEL
LIN {X 0,Y 632.739,Z 762.06,A -85,B 0,C 180,E1 6693.323,E2 6693.323} C_VEL
LIN {X 0,Y 632.646,Z 762.06,A -85,B 0,C 180,E1 6698.395,E2 6698.395} C_VEL
LIN {X 0,Y 632.595,Z 762.06,A -85,B 0,C 180,E1 6700.784,E2 6700.784} C_VEL
LIN {X 0,Y 628.697,Z 762.06,A -85,B 0,C 180,E1 6701.796,E2 6701.796} C_VEL
LIN {X 0,Y 624.775,Z 762.06,A -85,B 0,C 180,E1 6702.821,E2 6702.821} C_VEL
LIN {X 0,Y 624.827,Z 762.06,A -85,B 0,C 180,E1 6703.637,E2 6703.637} C_VEL
LIN {X 0,Y 627.294,Z 767.793,A -85,B 0,C 180,E1 6703.972,E2 6703.972} C_VEL
LIN {X 0,Y 656.294,Z 817.444,A -85,B 0,C 180,E1 6707.258,E2 6707.258} C_VEL
LIN {X 0,Y 654.187,Z 870.01,A -85,B 0,C 180,E1 6708.264,E2 6708.264} C_VEL
LIN {X 0,Y 651.04,Z 915.542,A -85,B 0,C 180,E1 6709.646,E2 6709.646} C_VEL
LIN {X 0,Y 646.803,Z 963.472,A -85,B 0,C 180,E1 6711.725,E2 6711.725} C_VEL
LIN {X 0,Y 642.436,Z 1006.966,A -85,B 0,C 180,E1 6714.222,E2 6714.222} C_VEL
LIN {X 0,Y 637.936,Z 1049.696,A -85,B 0,C 180,E1 6717.391,E2 6717.391} C_VEL
LIN {X 0,Y 634.029,Z 1086.35,A -85,B 0,C 180,E1 6720.798,E2 6720.798} C_VEL
LIN {X 0,Y 630.639,Z 1120.883,A -85,B 0,C 180,E1 6724.808,E2 6724.808} C_VEL
LIN {X 0,Y 628.291,Z 1148.491,A -85,B 0,C 180,E1 6728.852,E2 6728.852} C_VEL
LIN {X 0,Y 626.723,Z 1171.707,A -85,B 0,C 180,E1 6733.181,E2 6733.181} C_VEL
LIN {X 0,Y 625.889,Z 1188.882,A -85,B 0,C 180,E1 6737.449,E2 6737.449} C_VEL
LIN {X 0,Y 625.574,Z 1200.698,A -85,B 0,C 180,E1 6741.666,E2 6741.666} C_VEL
LIN {X 0,Y 625.491,Z 1207.677,A -85,B 0,C 180,E1 6745.843,E2 6745.843} C_VEL
LIN {X 0,Y 625.539,Z 1210,A -85,B 0,C 180,E1 6749.999,E2 6749.999} C_VEL
LIN {X 0,Y 625.49,Z 1207.679,A -85,B 0,C 180,E1 6754.156,E2 6754.156} C_VEL
LIN {X 0,Y 625.571,Z 1200.702,A -85,B 0,C 180,E1 6758.333,E2 6758.333} C_VEL
LIN {X 0,Y 625.866,Z 1188.888,A -85,B 0,C 180,E1 6762.55,E2 6762.55} C_VEL
LIN {X 0,Y 626.691,Z 1171.713,A -85,B 0,C 180,E1 6766.818,E2 6766.818} C_VEL
LIN {X 0,Y 628.31,Z 1148.497,A -85,B 0,C 180,E1 6771.146,E2 6771.146} C_VEL
LIN {X 0,Y 630.593,Z 1120.9,A -85,B 0,C 180,E1 6775.192,E2 6775.192} C_VEL
LIN {X 0,Y 634.014,Z 1086.386,A -85,B 0,C 180,E1 6779.199,E2 6779.199} C_VEL
LIN {X 0,Y 637.855,Z 1049.861,A -85,B 0,C 180,E1 6782.599,E2 6782.599} C_VEL
LIN {X 0,Y 642.496,Z 1006.863,A -85,B 0,C 180,E1 6785.783,E2 6785.783} C_VEL
LIN {X 0,Y 646.959,Z 962.438,A -85,B 0,C 180,E1 6788.322,E2 6788.322} C_VEL
LIN {X 0,Y 651.104,Z 915.873,A -85,B 0,C 180,E1 6790.334,E2 6790.334} C_VEL
LIN {X 0,Y 654.041,Z 873.639,A -85,B 0,C 180,E1 6791.646,E2 6791.646} C_VEL
LIN {X 0,Y 656.113,Z 827.571,A -85,B 0,C 180,E1 6792.581,E2 6792.581} C_VEL
LIN {X 0,Y 655.77,Z 816.957,A -85,B 0,C 180,E1 6792.792,E2 6792.792} C_VEL
LIN {X 0,Y 631.042,Z 773.765,A -85,B 0,C 180,E1 6795.585,E2 6795.585} C_VEL
LIN {X 0,Y 624.851,Z 763.043,A -85,B 0,C 180,E1 6796.336,E2 6796.336} C_VEL
LIN {X 0,Y 624.736,Z 762.06,A -85,B 0,C 180,E1 6796.521,E2 6796.521} C_VEL
LIN {X 0,Y 624.699,Z 762.06,A -85,B 0,C 180,E1 6801.025,E2 6801.025} C_VEL
LIN {X 0,Y 624.698,Z 762.06,A -85,B 0,C 180,E1 6806.191,E2 6806.191} C_VEL
LIN {X 0,Y 624.734,Z 762.06,A -85,B 0,C 180,E1 6811.063,E2 6811.063} C_VEL
LIN {X 0,Y 624.845,Z 762.06,A -85,B 0,C 180,E1 6815.719,E2 6815.719} C_VEL
LIN {X 0,Y 624.968,Z 762.06,A -85,B 0,C 180,E1 6820.556,E2 6820.556} C_VEL
LIN {X 0,Y 625.126,Z 762.06,A -85,B 0,C 180,E1 6826.005,E2 6826.005} C_VEL
LIN {X 0,Y 625.25,Z 762.06,A -85,B 0,C 180,E1 6831.655,E2 6831.655} C_VEL
LIN {X 0,Y 625.357,Z 762.06,A -85,B 0,C 180,E1 6837.222,E2 6837.222} C_VEL
LIN {X 0,Y 625.516,Z 762.06,A -85,B 0,C 180,E1 6842.761,E2 6842.761} C_VEL
LIN {X 0,Y 625.32,Z 762.06,A -85,B 0,C 180,E1 6848.328,E2 6848.328} C_VEL
LIN {X 0,Y 624.936,Z 762.06,A -85,B 0,C 180,E1 6853.983,E2 6853.983} C_VEL
LIN {X 0,Y 624.845,Z 762.06,A -85,B 0,C 180,E1 6859.779,E2 6859.779} C_VEL
LIN {X 0,Y 624.844,Z 762.06,A -85,B 0,C 180,E1 6864.263,E2 6864.263} C_VEL
LIN {X 0,Y 624.737,Z 762.06,A -85,B 0,C 180,E1 6869.454,E2 6869.454} C_VEL
LIN {X 0,Y 624.724,Z 762.06,A -85,B 0,C 180,E1 6874.675,E2 6874.675} C_VEL
LIN {X 0,Y 624.607,Z 762.06,A -85,B 0,C 180,E1 6879.271,E2 6879.271} C_VEL
LIN {X 0,Y 624.622,Z 762.06,A -85,B 0,C 180,E1 6884.041,E2 6884.041} C_VEL
LIN {X 0,Y 627.055,Z 767.75,A -85,B 0,C 180,E1 6884.366,E2 6884.366} C_VEL
LIN {X 0,Y 652.352,Z 811.15,A -85,B 0,C 180,E1 6887.336,E2 6887.336} C_VEL
LIN {X 0,Y 655.267,Z 818.606,A -85,B 0,C 180,E1 6887.74,E2 6887.74} C_VEL
LIN {X 0,Y 652.559,Z 866.999,A -85,B 0,C 180,E1 6888.983,E2 6888.983} C_VEL
LIN {X 0,Y 649.097,Z 909.511,A -85,B 0,C 180,E1 6890.568,E2 6890.568} C_VEL
LIN {X 0,Y 644.919,Z 954.043,A -85,B 0,C 180,E1 6892.789,E2 6892.789} C_VEL
LIN {X 0,Y 640.609,Z 995.149,A -85,B 0,C 180,E1 6895.437,E2 6895.437} C_VEL
LIN {X 0,Y 636.153,Z 1035.793,A -85,B 0,C 180,E1 6898.748,E2 6898.748} C_VEL
LIN {X 0,Y 632.415,Z 1071.098,A -85,B 0,C 180,E1 6902.352,E2 6902.352} C_VEL
LIN {X 0,Y 629.466,Z 1103.443,A -85,B 0,C 180,E1 6906.479,E2 6906.479} C_VEL
LIN {X 0,Y 627.419,Z 1129.182,A -85,B 0,C 180,E1 6910.661,E2 6910.661} C_VEL
LIN {X 0,Y 626.314,Z 1150.188,A -85,B 0,C 180,E1 6915.074,E2 6915.074} C_VEL
LIN {X 0,Y 625.768,Z 1163.551,A -85,B 0,C 180,E1 6918.862,E2 6918.862} C_VEL
LIN {X 0,Y 625.6,Z 1173.652,A -85,B 0,C 180,E1 6923.064,E2 6923.064} C_VEL
LIN {X 0,Y 625.449,Z 1178.967,A -85,B 0,C 180,E1 6927.231,E2 6927.231} C_VEL
LIN {X 0,Y 625.522,Z 1179.656,A -85,B 0,C 180,E1 6931.385,E2 6931.385} C_VEL
LIN {X 0,Y 625.599,Z 1175.843,A -85,B 0,C 180,E1 6935.545,E2 6935.545} C_VEL
LIN {X 0,Y 625.689,Z 1167.21,A -85,B 0,C 180,E1 6939.734,E2 6939.734} C_VEL
LIN {X 0,Y 626.144,Z 1153.534,A -85,B 0,C 180,E1 6943.966,E2 6943.966} C_VEL
LIN {X 0,Y 627.111,Z 1134.503,A -85,B 0,C 180,E1 6948.256,E2 6948.256} C_VEL
LIN {X 0,Y 628.887,Z 1110.234,A -85,B 0,C 180,E1 6952.412,E2 6952.412} C_VEL
LIN {X 0,Y 631.627,Z 1080.188,A -85,B 0,C 180,E1 6956.496,E2 6956.496} C_VEL
LIN {X 0,Y 635.192,Z 1044.809,A -85,B 0,C 180,E1 6960.31,E2 6960.31} C_VEL
LIN {X 0,Y 639.363,Z 1006.089,A -85,B 0,C 180,E1 6963.661,E2 6963.661} C_VEL
LIN {X 0,Y 644.112,Z 961.247,A -85,B 0,C 180,E1 6966.707,E2 6966.707} C_VEL
LIN {X 0,Y 648.488,Z 917.403,A -85,B 0,C 180,E1 6968.989,E2 6968.989} C_VEL
LIN {X 0,Y 651.959,Z 874.582,A -85,B 0,C 180,E1 6970.675,E2 6970.675} C_VEL
LIN {X 0,Y 654.675,Z 831.435,A -85,B 0,C 180,E1 6971.895,E2 6971.895} C_VEL
LIN {X 0,Y 654.787,Z 816.755,A -85,B 0,C 180,E1 6972.251,E2 6972.251} C_VEL
LIN {X 0,Y 633.372,Z 777.79,A -85,B 0,C 180,E1 6974.801,E2 6974.801} C_VEL
LIN {X 0,Y 624.833,Z 763.02,A -85,B 0,C 180,E1 6975.831,E2 6975.831} C_VEL
LIN {X 0,Y 624.751,Z 762.06,A -85,B 0,C 180,E1 6976.032,E2 6976.032} C_VEL
LIN {X 0,Y 624.664,Z 762.06,A -85,B 0,C 180,E1 6981.043,E2 6981.043} C_VEL
LIN {X 0,Y 624.672,Z 762.06,A -85,B 0,C 180,E1 6986.209,E2 6986.209} C_VEL
LIN {X 0,Y 624.676,Z 762.06,A -85,B 0,C 180,E1 6991.079,E2 6991.079} C_VEL
LIN {X 0,Y 624.726,Z 762.06,A -85,B 0,C 180,E1 6995.732,E2 6995.732} C_VEL
LIN {X 0,Y 624.768,Z 762.06,A -85,B 0,C 180,E1 7000.613,E2 7000.613} C_VEL
LIN {X 0,Y 624.953,Z 762.06,A -85,B 0,C 180,E1 7006.018,E2 7006.018} C_VEL
LIN {X 0,Y 625.335,Z 762.06,A -85,B 0,C 180,E1 7011.673,E2 7011.673} C_VEL
LIN {X 0,Y 625.522,Z 762.06,A -85,B 0,C 180,E1 7017.239,E2 7017.239} C_VEL
LIN {X 0,Y 625.555,Z 762.06,A -85,B 0,C 180,E1 7021.392,E2 7021.392} C_VEL
LIN {X 0,Y 625.238,Z 762.06,A -85,B 0,C 180,E1 7026.948,E2 7026.948} C_VEL
LIN {X 0,Y 625.154,Z 762.06,A -85,B 0,C 180,E1 7032.572,E2 7032.572} C_VEL
LIN {X 0,Y 625.128,Z 762.06,A -85,B 0,C 180,E1 7038.321,E2 7038.321} C_VEL
LIN {X 0,Y 624.945,Z 762.06,A -85,B 0,C 180,E1 7043.242,E2 7043.242} C_VEL
LIN {X 0,Y 624.855,Z 762.06,A -85,B 0,C 180,E1 7048.93,E2 7048.93} C_VEL
LIN {X 0,Y 624.765,Z 762.06,A -85,B 0,C 180,E1 7053.805,E2 7053.805} C_VEL
LIN {X 0,Y 624.675,Z 762.06,A -85,B 0,C 180,E1 7059.276,E2 7059.276} C_VEL
LIN {X 0,Y 624.775,Z 762.06,A -85,B 0,C 180,E1 7062.821,E2 7062.821} C_VEL
LIN {X 0,Y 625.277,Z 765.484,A -85,B 0,C 180,E1 7063.497,E2 7063.497} C_VEL
LIN {X 0,Y 627.709,Z 776.798,A -85,B 0,C 180,E1 7064.155,E2 7064.155} C_VEL
LIN {X 0,Y 632.279,Z 788.921,A -85,B 0,C 180,E1 7064.768,E2 7064.768} C_VEL
LIN {X 0,Y 650.482,Z 821.66,A -85,B 0,C 180,E1 7066.858,E2 7066.858} C_VEL
LIN {X 0,Y 648.024,Z 873.407,A -85,B 0,C 180,E1 7067.873,E2 7067.873} C_VEL
LIN {X 0,Y 644.568,Z 919.235,A -85,B 0,C 180,E1 7069.325,E2 7069.325} C_VEL
LIN {X 0,Y 640.034,Z 968.048,A -85,B 0,C 180,E1 7071.507,E2 7071.507} C_VEL
LIN {X 0,Y 635.161,Z 1011.984,A -85,B 0,C 180,E1 7074.129,E2 7074.129} C_VEL
LIN {X 0,Y 630.515,Z 1053.776,A -85,B 0,C 180,E1 7077.324,E2 7077.324} C_VEL
LIN {X 0,Y 626.129,Z 1091.828,A -85,B 0,C 180,E1 7081.012,E2 7081.012} C_VEL
LIN {X 0,Y 622.896,Z 1123.806,A -85,B 0,C 180,E1 7084.878,E2 7084.878} C_VEL
LIN {X 0,Y 620.257,Z 1152.877,A -85,B 0,C 180,E1 7089.32,E2 7089.32} C_VEL
LIN {X 0,Y 618.847,Z 1173.373,A -85,B 0,C 180,E1 7093.326,E2 7093.326} C_VEL
LIN {X 0,Y 617.989,Z 1190.233,A -85,B 0,C 180,E1 7097.707,E2 7097.707} C_VEL
LIN {X 0,Y 617.689,Z 1201.926,A -85,B 0,C 180,E1 7102.125,E2 7102.125} C_VEL
LIN {X 0,Y 617.587,Z 1207.677,A -85,B 0,C 180,E1 7105.79,E2 7105.79} C_VEL
LIN {X 0,Y 617.659,Z 1210,A -85,B 0,C 180,E1 7109.999,E2 7109.999} C_VEL
LIN {X 0,Y 617.586,Z 1207.679,A -85,B 0,C 180,E1 7114.209,E2 7114.209} C_VEL
LIN {X 0,Y 617.678,Z 1200.699,A -85,B 0,C 180,E1 7118.44,E2 7118.44} C_VEL
LIN {X 0,Y 618.02,Z 1188.888,A -85,B 0,C 180,E1 7122.712,E2 7122.712} C_VEL
LIN {X 0,Y 618.931,Z 1171.711,A -85,B 0,C 180,E1 7127.036,E2 7127.036} C_VEL
LIN {X 0,Y 620.629,Z 1148.499,A -85,B 0,C 180,E1 7131.42,E2 7131.42} C_VEL
LIN {X 0,Y 623.103,Z 1121.052,A -85,B 0,C 180,E1 7135.496,E2 7135.496} C_VEL
LIN {X 0,Y 626.873,Z 1085.368,A -85,B 0,C 180,E1 7139.679,E2 7139.679} C_VEL
LIN {X 0,Y 631.083,Z 1048.29,A -85,B 0,C 180,E1 7143.133,E2 7143.133} C_VEL
LIN {X 0,Y 636,Z 1005.796,A -85,B 0,C 180,E1 7146.286,E2 7146.286} C_VEL
LIN {X 0,Y 640.784,Z 960.761,A -85,B 0,C 180,E1 7148.855,E2 7148.855} C_VEL
LIN {X 0,Y 645.131,Z 913.926,A -85,B 0,C 180,E1 7150.871,E2 7150.871} C_VEL
LIN {X 0,Y 648.365,Z 867.346,A -85,B 0,C 180,E1 7152.273,E2 7152.273} C_VEL
LIN {X 0,Y 649.86,Z 820.001,A -85,B 0,C 180,E1 7153.223,E2 7153.223} C_VEL
LIN {X 0,Y 626.371,Z 779.052,A -85,B 0,C 180,E1 7155.934,E2 7155.934} C_VEL
LIN {X 0,Y 616.906,Z 763.15,A -85,B 0,C 180,E1 7157.107,E2 7157.107} C_VEL
LIN {X 0,Y 616.849,Z 762.06,A -85,B 0,C 180,E1 7157.299,E2 7157.299} C_VEL
LIN {X 0,Y 616.755,Z 762.06,A -85,B 0,C 180,E1 7162.223,E2 7162.223} C_VEL
LIN {X 0,Y 616.756,Z 762.06,A -85,B 0,C 180,E1 7167.378,E2 7167.378} C_VEL
LIN {X 0,Y 616.823,Z 762.06,A -85,B 0,C 180,E1 7172.254,E2 7172.254} C_VEL
LIN {X 0,Y 616.915,Z 762.06,A -85,B 0,C 180,E1 7176.921,E2 7176.921} C_VEL
LIN {X 0,Y 617.116,Z 762.06,A -85,B 0,C 180,E1 7182.74,E2 7182.74} C_VEL
LIN {X 0,Y 617.218,Z 762.06,A -85,B 0,C 180,E1 7188.32,E2 7188.32} C_VEL
LIN {X 0,Y 617.331,Z 762.06,A -85,B 0,C 180,E1 7192.963,E2 7192.963} C_VEL
LIN {X 0,Y 617.64,Z 762.06,A -85,B 0,C 180,E1 7198.59,E2 7198.59} C_VEL
LIN {X 0,Y 617.508,Z 762.06,A -85,B 0,C 180,E1 7204.201,E2 7204.201} C_VEL
LIN {X 0,Y 617.282,Z 762.06,A -85,B 0,C 180,E1 7209.857,E2 7209.857} C_VEL
LIN {X 0,Y 616.945,Z 762.06,A -85,B 0,C 180,E1 7215.62,E2 7215.62} C_VEL
LIN {X 0,Y 616.938,Z 762.06,A -85,B 0,C 180,E1 7221.544,E2 7221.544} C_VEL
LIN {X 0,Y 616.886,Z 762.06,A -85,B 0,C 180,E1 7226.15,E2 7226.15} C_VEL
LIN {X 0,Y 616.855,Z 762.06,A -85,B 0,C 180,E1 7230.976,E2 7230.976} C_VEL
LIN {X 0,Y 616.776,Z 762.06,A -85,B 0,C 180,E1 7236.051,E2 7236.051} C_VEL
LIN {X 0,Y 616.69,Z 762.06,A -85,B 0,C 180,E1 7241.404,E2 7241.404} C_VEL
LIN {X 0,Y 616.668,Z 762.06,A -85,B 0,C 180,E1 7243.264,E2 7243.264} C_VEL
LIN {X 0,Y 618.945,Z 767.576,A -85,B 0,C 180,E1 7243.585,E2 7243.585} C_VEL
LIN {X 0,Y 644.422,Z 810.61,A -85,B 0,C 180,E1 7246.672,E2 7246.672} C_VEL
LIN {X 0,Y 649.272,Z 820.259,A -85,B 0,C 180,E1 7247.297,E2 7247.297} C_VEL
LIN {X 0,Y 646.476,Z 867.58,A -85,B 0,C 180,E1 7248.536,E2 7248.536} C_VEL
LIN {X 0,Y 642.885,Z 909.493,A -85,B 0,C 180,E1 7250.111,E2 7250.111} C_VEL
LIN {X 0,Y 638.414,Z 954.034,A -85,B 0,C 180,E1 7252.345,E2 7252.345} C_VEL
LIN {X 0,Y 633.917,Z 994.22,A -85,B 0,C 180,E1 7254.943,E2 7254.943} C_VEL
LIN {X 0,Y 629.084,Z 1035.786,A -85,B 0,C 180,E1 7258.357,E2 7258.357} C_VEL
LIN {X 0,Y 625.076,Z 1071.374,A -85,B 0,C 180,E1 7262.033,E2 7262.033} C_VEL
LIN {X 0,Y 621.882,Z 1103.437,A -85,B 0,C 180,E1 7266.174,E2 7266.174} C_VEL
LIN {X 0,Y 619.698,Z 1129.18,A -85,B 0,C 180,E1 7270.411,E2 7270.411} C_VEL
LIN {X 0,Y 618.484,Z 1149.273,A -85,B 0,C 180,E1 7274.665,E2 7274.665} C_VEL
LIN {X 0,Y 617.885,Z 1163.55,A -85,B 0,C 180,E1 7278.718,E2 7278.718} C_VEL
LIN {X 0,Y 617.715,Z 1173.648,A -85,B 0,C 180,E1 7282.975,E2 7282.975} C_VEL
LIN {X 0,Y 617.566,Z 1178.963,A -85,B 0,C 180,E1 7287.196,E2 7287.196} C_VEL
LIN {X 0,Y 617.643,Z 1179.656,A -85,B 0,C 180,E1 7291.403,E2 7291.403} C_VEL
LIN {X 0,Y 617.714,Z 1175.844,A -85,B 0,C 180,E1 7295.616,E2 7295.616} C_VEL
LIN {X 0,Y 617.797,Z 1167.212,A -85,B 0,C 180,E1 7299.859,E2 7299.859} C_VEL
LIN {X 0,Y 618.317,Z 1153.537,A -85,B 0,C 180,E1 7304.147,E2 7304.147} C_VEL
LIN {X 0,Y 619.368,Z 1134.508,A -85,B 0,C 180,E1 7308.493,E2 7308.493} C_VEL
LIN {X 0,Y 621.226,Z 1110.796,A -85,B 0,C 180,E1 7312.615,E2 7312.615} C_VEL
LIN {X 0,Y 624.188,Z 1080.548,A -85,B 0,C 180,E1 7316.791,E2 7316.791} C_VEL
LIN {X 0,Y 628.034,Z 1045.212,A -85,B 0,C 180,E1 7320.651,E2 7320.651} C_VEL
LIN {X 0,Y 632.41,Z 1007.251,A -85,B 0,C 180,E1 7323.986,E2 7323.986} C_VEL
LIN {X 0,Y 637.32,Z 963.506,A -85,B 0,C 180,E1 7327.007,E2 7327.007} C_VEL
LIN {X 0,Y 641.881,Z 921.208,A -85,B 0,C 180,E1 7329.272,E2 7329.272} C_VEL
LIN {X 0,Y 645.618,Z 878.337,A -85,B 0,C 180,E1 7331.012,E2 7331.012} C_VEL
LIN {X 0,Y 648.631,Z 833.37,A -85,B 0,C 180,E1 7332.32,E2 7332.32} C_VEL
LIN {X 0,Y 648.808,Z 819.925,A -85,B 0,C 180,E1 7332.659,E2 7332.659} C_VEL
LIN {X 0,Y 626.824,Z 779.621,A -85,B 0,C 180,E1 7335.375,E2 7335.375} C_VEL
LIN {X 0,Y 616.864,Z 763.241,A -85,B 0,C 180,E1 7336.602,E2 7336.602} C_VEL
LIN {X 0,Y 616.781,Z 762.06,A -85,B 0,C 180,E1 7336.704,E2 7336.704} C_VEL
LIN {X 0,Y 616.736,Z 762.06,A -85,B 0,C 180,E1 7342.242,E2 7342.242} C_VEL
LIN {X 0,Y 616.755,Z 762.06,A -85,B 0,C 180,E1 7347.397,E2 7347.397} C_VEL
LIN {X 0,Y 616.758,Z 762.06,A -85,B 0,C 180,E1 7352.269,E2 7352.269} C_VEL
LIN {X 0,Y 616.813,Z 762.06,A -85,B 0,C 180,E1 7356.934,E2 7356.934} C_VEL
LIN {X 0,Y 616.821,Z 762.06,A -85,B 0,C 180,E1 7361.44,E2 7361.44} C_VEL
LIN {X 0,Y 617.146,Z 762.06,A -85,B 0,C 180,E1 7367.279,E2 7367.279} C_VEL
LIN {X 0,Y 617.44,Z 762.06,A -85,B 0,C 180,E1 7372.98,E2 7372.98} C_VEL
LIN {X 0,Y 617.562,Z 762.06,A -85,B 0,C 180,E1 7378.606,E2 7378.606} C_VEL
LIN {X 0,Y 617.468,Z 762.06,A -85,B 0,C 180,E1 7382.813,E2 7382.813} C_VEL
LIN {X 0,Y 617.349,Z 762.06,A -85,B 0,C 180,E1 7388.452,E2 7388.452} C_VEL
LIN {X 0,Y 617.221,Z 762.06,A -85,B 0,C 180,E1 7394.178,E2 7394.178} C_VEL
LIN {X 0,Y 617.214,Z 762.06,A -85,B 0,C 180,E1 7398.565,E2 7398.565} C_VEL
LIN {X 0,Y 617.056,Z 762.06,A -85,B 0,C 180,E1 7403.074,E2 7403.074} C_VEL
LIN {X 0,Y 616.949,Z 762.06,A -85,B 0,C 180,E1 7408.143,E2 7408.143} C_VEL
LIN {X 0,Y 616.845,Z 762.06,A -85,B 0,C 180,E1 7413.6,E2 7413.6} C_VEL
LIN {X 0,Y 616.749,Z 762.06,A -85,B 0,C 180,E1 7418.367,E2 7418.367} C_VEL
LIN {X 0,Y 616.897,Z 762.06,A -85,B 0,C 180,E1 7422.858,E2 7422.858} C_VEL
LIN {X 0,Y 619.306,Z 767.765,A -85,B 0,C 180,E1 7423.206,E2 7423.206} C_VEL
LIN {X 0,Y 632.279,Z 788.921,A -85,B 0,C 180,E1 7424.768,E2 7424.768} C_VEL
LIN {X 0,Y 634.474,Z 796.745,A -85,B 0,C 180,E1 7425.088,E2 7425.088} C_VEL
LIN {X 0,Y 636.611,Z 809.347,A -85,B 0,C 180,E1 7425.473,E2 7425.473} C_VEL
LIN {X 0,Y 637.217,Z 810.452,A -85,B 0,C 180,E1 7425.543,E2 7425.543} C_VEL
LIN {X 0,Y 644.639,Z 824.999,A -85,B 0,C 180,E1 7426.43,E2 7426.43} C_VEL
LIN {X 0,Y 642.006,Z 875.636,A -85,B 0,C 180,E1 7427.453,E2 7427.453} C_VEL
LIN {X 0,Y 638.167,Z 922.888,A -85,B 0,C 180,E1 7428.998,E2 7428.998} C_VEL
LIN {X 0,Y 633.545,Z 969.589,A -85,B 0,C 180,E1 7431.129,E2 7431.129} C_VEL
LIN {X 0,Y 628.308,Z 1013.728,A -85,B 0,C 180,E1 7433.81,E2 7433.81} C_VEL
LIN {X 0,Y 623.538,Z 1054.291,A -85,B 0,C 180,E1 7436.96,E2 7436.96} C_VEL
LIN {X 0,Y 618.778,Z 1092.942,A -85,B 0,C 180,E1 7440.763,E2 7440.763} C_VEL
LIN {X 0,Y 615.274,Z 1125.151,A -85,B 0,C 180,E1 7444.739,E2 7444.739} C_VEL
LIN {X 0,Y 612.513,Z 1153.922,A -85,B 0,C 180,E1 7449.229,E2 7449.229} C_VEL
LIN {X 0,Y 610.927,Z 1174.925,A -85,B 0,C 180,E1 7453.473,E2 7453.473} C_VEL
LIN {X 0,Y 610.099,Z 1191.135,A -85,B 0,C 180,E1 7457.833,E2 7457.833} C_VEL
LIN {X 0,Y 609.807,Z 1201.944,A -85,B 0,C 180,E1 7462.032,E2 7462.032} C_VEL
LIN {X 0,Y 609.683,Z 1207.677,A -85,B 0,C 180,E1 7465.735,E2 7465.735} C_VEL
LIN {X 0,Y 609.758,Z 1210,A -85,B 0,C 180,E1 7469.999,E2 7469.999} C_VEL
LIN {X 0,Y 609.682,Z 1207.68,A -85,B 0,C 180,E1 7474.263,E2 7474.263} C_VEL
LIN {X 0,Y 609.792,Z 1200.696,A -85,B 0,C 180,E1 7478.55,E2 7478.55} C_VEL
LIN {X 0,Y 610.172,Z 1188.888,A -85,B 0,C 180,E1 7482.878,E2 7482.878} C_VEL
LIN {X 0,Y 611.194,Z 1171.71,A -85,B 0,C 180,E1 7487.258,E2 7487.258} C_VEL
LIN {X 0,Y 613.081,Z 1147.17,A -85,B 0,C 180,E1 7491.927,E2 7491.927} C_VEL
LIN {X 0,Y 615.818,Z 1119.594,A -85,B 0,C 180,E1 7496.015,E2 7496.015} C_VEL
LIN {X 0,Y 619.889,Z 1084.006,A -85,B 0,C 180,E1 7500.204,E2 7500.204} C_VEL
LIN {X 0,Y 624.557,Z 1045.119,A -85,B 0,C 180,E1 7503.812,E2 7503.812} C_VEL
LIN {X 0,Y 629.443,Z 1005.102,A -85,B 0,C 180,E1 7506.776,E2 7506.776} C_VEL
LIN {X 0,Y 634.585,Z 959.678,A -85,B 0,C 180,E1 7509.371,E2 7509.371} C_VEL
LIN {X 0,Y 639.099,Z 913.124,A -85,B 0,C 180,E1 7511.374,E2 7511.374} C_VEL
LIN {X 0,Y 642.578,Z 866.06,A -85,B 0,C 180,E1 7512.78,E2 7512.78} C_VEL
LIN {X 0,Y 644.263,Z 823.638,A -85,B 0,C 180,E1 7513.626,E2 7513.626} C_VEL
LIN {X 0,Y 621.516,Z 783.959,A -85,B 0,C 180,E1 7516.314,E2 7516.314} C_VEL
LIN {X 0,Y 609.043,Z 763.567,A -85,B 0,C 180,E1 7517.895,E2 7517.895} C_VEL
LIN {X 0,Y 608.922,Z 762.06,A -85,B 0,C 180,E1 7518.046,E2 7518.046} C_VEL
LIN {X 0,Y 608.847,Z 762.06,A -85,B 0,C 180,E1 7523.435,E2 7523.435} C_VEL
LIN {X 0,Y 608.84,Z 762.06,A -85,B 0,C 180,E1 7528.581,E2 7528.581} C_VEL
LIN {X 0,Y 608.94,Z 762.06,A -85,B 0,C 180,E1 7533.464,E2 7533.464} C_VEL
LIN {X 0,Y 609.014,Z 762.06,A -85,B 0,C 180,E1 7538.144,E2 7538.144} C_VEL
LIN {X 0,Y 609.217,Z 762.06,A -85,B 0,C 180,E1 7542.677,E2 7542.677} C_VEL
LIN {X 0,Y 609.299,Z 762.06,A -85,B 0,C 180,E1 7547.096,E2 7547.096} C_VEL
LIN {X 0,Y 609.42,Z 762.06,A -85,B 0,C 180,E1 7552.871,E2 7552.871} C_VEL
LIN {X 0,Y 609.733,Z 762.06,A -85,B 0,C 180,E1 7558.572,E2 7558.572} C_VEL
LIN {X 0,Y 609.598,Z 762.06,A -85,B 0,C 180,E1 7564.256,E2 7564.256} C_VEL
LIN {X 0,Y 609.362,Z 762.06,A -85,B 0,C 180,E1 7569.987,E2 7569.987} C_VEL
LIN {X 0,Y 609.017,Z 762.06,A -85,B 0,C 180,E1 7575.828,E2 7575.828} C_VEL
LIN {X 0,Y 609.001,Z 762.06,A -85,B 0,C 180,E1 7581.839,E2 7581.839} C_VEL
LIN {X 0,Y 608.922,Z 762.06,A -85,B 0,C 180,E1 7586.7,E2 7586.7} C_VEL
LIN {X 0,Y 608.919,Z 762.06,A -85,B 0,C 180,E1 7592.463,E2 7592.463} C_VEL
LIN {X 0,Y 608.833,Z 762.06,A -85,B 0,C 180,E1 7598.336,E2 7598.336} C_VEL
LIN {X 0,Y 608.788,Z 762.141,A -85,B 0,C 180,E1 7602.471,E2 7602.471} C_VEL
LIN {X 0,Y 611.301,Z 767.834,A -85,B 0,C 180,E1 7602.826,E2 7602.826} C_VEL
LIN {X 0,Y 636.982,Z 810.973,A -85,B 0,C 180,E1 7606.048,E2 7606.048} C_VEL
LIN {X 0,Y 643.327,Z 823.917,A -85,B 0,C 180,E1 7606.893,E2 7606.893} C_VEL
LIN {X 0,Y 640.028,Z 872.543,A -85,B 0,C 180,E1 7608.227,E2 7608.227} C_VEL
LIN {X 0,Y 635.909,Z 917.737,A -85,B 0,C 180,E1 7610.014,E2 7610.014} C_VEL
LIN {X 0,Y 631.353,Z 959.699,A -85,B 0,C 180,E1 7612.224,E2 7612.224} C_VEL
LIN {X 0,Y 626.112,Z 1003.111,A -85,B 0,C 180,E1 7615.187,E2 7615.187} C_VEL
LIN {X 0,Y 621.492,Z 1040.74,A -85,B 0,C 180,E1 7618.425,E2 7618.425} C_VEL
LIN {X 0,Y 617.056,Z 1077.583,A -85,B 0,C 180,E1 7622.409,E2 7622.409} C_VEL
LIN {X 0,Y 613.958,Z 1107.314,A -85,B 0,C 180,E1 7626.457,E2 7626.457} C_VEL
LIN {X 0,Y 611.696,Z 1133.066,A -85,B 0,C 180,E1 7630.894,E2 7630.894} C_VEL
LIN {X 0,Y 610.582,Z 1152.222,A -85,B 0,C 180,E1 7635.222,E2 7635.222} C_VEL
LIN {X 0,Y 609.991,Z 1165.533,A -85,B 0,C 180,E1 7639.293,E2 7639.293} C_VEL
LIN {X 0,Y 609.839,Z 1174.852,A -85,B 0,C 180,E1 7643.599,E2 7643.599} C_VEL
LIN {X 0,Y 609.66,Z 1178.96,A -85,B 0,C 180,E1 7647.159,E2 7647.159} C_VEL
LIN {X 0,Y 609.739,Z 1179.656,A -85,B 0,C 180,E1 7651.421,E2 7651.421} C_VEL
LIN {X 0,Y 609.808,Z 1175.845,A -85,B 0,C 180,E1 7655.689,E2 7655.689} C_VEL
LIN {X 0,Y 609.905,Z 1167.211,A -85,B 0,C 180,E1 7659.988,E2 7659.988} C_VEL
LIN {X 0,Y 610.5,Z 1153.54,A -85,B 0,C 180,E1 7664.332,E2 7664.332} C_VEL
LIN {X 0,Y 611.63,Z 1134.512,A -85,B 0,C 180,E1 7668.735,E2 7668.735} C_VEL
LIN {X 0,Y 613.642,Z 1110.796,A -85,B 0,C 180,E1 7672.911,E2 7672.911} C_VEL
LIN {X 0,Y 616.9,Z 1080.058,A -85,B 0,C 180,E1 7677.199,E2 7677.199} C_VEL
LIN {X 0,Y 621.018,Z 1044.318,A -85,B 0,C 180,E1 7681.131,E2 7681.131} C_VEL
LIN {X 0,Y 625.691,Z 1006.648,A -85,B 0,C 180,E1 7684.453,E2 7684.453} C_VEL
LIN {X 0,Y 630.93,Z 962.299,A -85,B 0,C 180,E1 7687.531,E2 7687.531} C_VEL
LIN {X 0,Y 635.818,Z 918.746,A -85,B 0,C 180,E1 7689.85,E2 7689.85} C_VEL
LIN {X 0,Y 639.726,Z 876.744,A -85,B 0,C 180,E1 7691.537,E2 7691.537} C_VEL
LIN {X 0,Y 642.798,Z 833.376,A -85,B 0,C 180,E1 7692.795,E2 7692.795} C_VEL
LIN {X 0,Y 642.889,Z 823.058,A -85,B 0,C 180,E1 7693.073,E2 7693.073} C_VEL
LIN {X 0,Y 621.879,Z 784.464,A -85,B 0,C 180,E1 7695.764,E2 7695.764} C_VEL
LIN {X 0,Y 608.982,Z 763.375,A -85,B 0,C 180,E1 7697.398,E2 7697.398} C_VEL
LIN {X 0,Y 608.868,Z 762.06,A -85,B 0,C 180,E1 7697.468,E2 7697.468} C_VEL
LIN {X 0,Y 608.822,Z 762.06,A -85,B 0,C 180,E1 7702.585,E2 7702.585} C_VEL
LIN {X 0,Y 608.845,Z 762.06,A -85,B 0,C 180,E1 7708.601,E2 7708.601} C_VEL
LIN {X 0,Y 608.857,Z 762.06,A -85,B 0,C 180,E1 7713.478,E2 7713.478} C_VEL
LIN {X 0,Y 608.914,Z 762.06,A -85,B 0,C 180,E1 7718.158,E2 7718.158} C_VEL
LIN {X 0,Y 609.034,Z 762.06,A -85,B 0,C 180,E1 7724.172,E2 7724.172} C_VEL
LIN {X 0,Y 609.378,Z 762.06,A -85,B 0,C 180,E1 7730.013,E2 7730.013} C_VEL
LIN {X 0,Y 609.501,Z 762.06,A -85,B 0,C 180,E1 7734.318,E2 7734.318} C_VEL
LIN {X 0,Y 609.662,Z 762.06,A -85,B 0,C 180,E1 7738.588,E2 7738.588} C_VEL
LIN {X 0,Y 609.565,Z 762.06,A -85,B 0,C 180,E1 7742.85,E2 7742.85} C_VEL
LIN {X 0,Y 609.436,Z 762.06,A -85,B 0,C 180,E1 7748.563,E2 7748.563} C_VEL
LIN {X 0,Y 609.297,Z 762.06,A -85,B 0,C 180,E1 7754.366,E2 7754.366} C_VEL
LIN {X 0,Y 609.249,Z 762.06,A -85,B 0,C 180,E1 7759.521,E2 7759.521} C_VEL
LIN {X 0,Y 609.136,Z 762.06,A -85,B 0,C 180,E1 7764.949,E2 7764.949} C_VEL
LIN {X 0,Y 609.021,Z 762.06,A -85,B 0,C 180,E1 7769.757,E2 7769.757} C_VEL
LIN {X 0,Y 608.881,Z 762.06,A -85,B 0,C 180,E1 7775.015,E2 7775.015} C_VEL
LIN {X 0,Y 608.872,Z 762.06,A -85,B 0,C 180,E1 7780.191,E2 7780.191} C_VEL
LIN {X 0,Y 608.96,Z 762.114,A -85,B 0,C 180,E1 7782.071,E2 7782.071} C_VEL
LIN {X 0,Y 611.195,Z 767.57,A -85,B 0,C 180,E1 7782.394,E2 7782.394} C_VEL
LIN {X 0,Y 635.999,Z 808.494,A -85,B 0,C 180,E1 7785.406,E2 7785.406} C_VEL
LIN {X 0,Y 637.217,Z 810.452,A -85,B 0,C 180,E1 7785.543,E2 7785.543} C_VEL
LIN {X 0,Y 639.91,Z 819.94,A -85,B 0,C 180,E1 7785.933,E2 7785.933} C_VEL
LIN {X 0,Y 638.156,Z 844.941,A -85,B 0,C 180,E1 7786.289,E2 7786.289} C_VEL
LIN {X 0,Y 634.87,Z 892.003,A -85,B 0,C 180,E1 7787.439,E2 7787.439} C_VEL
LIN {X 0,Y 631.009,Z 935.647,A -85,B 0,C 180,E1 7789.046,E2 7789.046} C_VEL
LIN {X 0,Y 625.982,Z 980.502,A -85,B 0,C 180,E1 7791.278,E2 7791.278} C_VEL
LIN {X 0,Y 620.714,Z 1022.674,A -85,B 0,C 180,E1 7793.999,E2 7793.999} C_VEL
LIN {X 0,Y 615.322,Z 1063.651,A -85,B 0,C 180,E1 7797.397,E2 7797.397} C_VEL
LIN {X 0,Y 610.788,Z 1099.303,A -85,B 0,C 180,E1 7801.105,E2 7801.105} C_VEL
LIN {X 0,Y 606.907,Z 1132.24,A -85,B 0,C 180,E1 7805.418,E2 7805.418} C_VEL
LIN {X 0,Y 604.544,Z 1156.966,A -85,B 0,C 180,E1 7809.515,E2 7809.515} C_VEL
LIN {X 0,Y 602.941,Z 1178.003,A -85,B 0,C 180,E1 7813.996,E2 7813.996} C_VEL
LIN {X 0,Y 602.192,Z 1193.417,A -85,B 0,C 180,E1 7818.419,E2 7818.419} C_VEL
LIN {X 0,Y 601.885,Z 1203.563,A -85,B 0,C 180,E1 7822.788,E2 7822.788} C_VEL
LIN {X 0,Y 601.871,Z 1208.923,A -85,B 0,C 180,E1 7827.121,E2 7827.121} C_VEL
LIN {X 0,Y 602.039,Z 1209.667,A -85,B 0,C 180,E1 7831.438,E2 7831.438} C_VEL
LIN {X 0,Y 601.855,Z 1205.912,A -85,B 0,C 180,E1 7835.763,E2 7835.763} C_VEL
LIN {X 0,Y 602.073,Z 1197.331,A -85,B 0,C 180,E1 7840.118,E2 7840.118} C_VEL
LIN {X 0,Y 602.713,Z 1183.713,A -85,B 0,C 180,E1 7844.519,E2 7844.519} C_VEL
LIN {X 0,Y 603.944,Z 1164.729,A -85,B 0,C 180,E1 7848.981,E2 7848.981} C_VEL
LIN {X 0,Y 606.224,Z 1139.246,A -85,B 0,C 180,E1 7853.504,E2 7853.504} C_VEL
LIN {X 0,Y 609.62,Z 1109.307,A -85,B 0,C 180,E1 7857.694,E2 7857.694} C_VEL
LIN {X 0,Y 614.139,Z 1072.568,A -85,B 0,C 180,E1 7861.754,E2 7861.754} C_VEL
LIN {X 0,Y 619.178,Z 1034.157,A -85,B 0,C 180,E1 7865.126,E2 7865.126} C_VEL
LIN {X 0,Y 624.7,Z 990.983,A -85,B 0,C 180,E1 7868.112,E2 7868.112} C_VEL
LIN {X 0,Y 629.79,Z 946.848,A -85,B 0,C 180,E1 7870.455,E2 7870.455} C_VEL
LIN {X 0,Y 634.328,Z 898.191,A -85,B 0,C 180,E1 7872.368,E2 7872.368} C_VEL
LIN {X 0,Y 637.728,Z 849.477,A -85,B 0,C 180,E1 7873.639,E2 7873.639} C_VEL
LIN {X 0,Y 638.205,Z 826.419,A -85,B 0,C 180,E1 7874.096,E2 7874.096} C_VEL
LIN {X 0,Y 616.255,Z 788.088,A -85,B 0,C 180,E1 7876.756,E2 7876.756} C_VEL
LIN {X 0,Y 601.086,Z 763.46,A -85,B 0,C 180,E1 7878.737,E2 7878.737} C_VEL
LIN {X 0,Y 600.942,Z 762.06,A -85,B 0,C 180,E1 7878.823,E2 7878.823} C_VEL
LIN {X 0,Y 600.92,Z 762.06,A -85,B 0,C 180,E1 7884.659,E2 7884.659} C_VEL
LIN {X 0,Y 600.93,Z 762.06,A -85,B 0,C 180,E1 7889.801,E2 7889.801} C_VEL
LIN {X 0,Y 601.068,Z 762.06,A -85,B 0,C 180,E1 7894.829,E2 7894.829} C_VEL
LIN {X 0,Y 601.118,Z 762.06,A -85,B 0,C 180,E1 7899.388,E2 7899.388} C_VEL
LIN {X 0,Y 601.325,Z 762.06,A -85,B 0,C 180,E1 7903.946,E2 7903.946} C_VEL
LIN {X 0,Y 601.46,Z 762.06,A -85,B 0,C 180,E1 7909.864,E2 7909.864} C_VEL
LIN {X 0,Y 601.695,Z 762.06,A -85,B 0,C 180,E1 7915.671,E2 7915.671} C_VEL
LIN {X 0,Y 601.847,Z 762.06,A -85,B 0,C 180,E1 7919.992,E2 7919.992} C_VEL
LIN {X 0,Y 601.701,Z 762.06,A -85,B 0,C 180,E1 7924.312,E2 7924.312} C_VEL
LIN {X 0,Y 601.568,Z 762.06,A -85,B 0,C 180,E1 7928.659,E2 7928.659} C_VEL
LIN {X 0,Y 601.264,Z 762.06,A -85,B 0,C 180,E1 7933.063,E2 7933.063} C_VEL
LIN {X 0,Y 601.027,Z 762.06,A -85,B 0,C 180,E1 7939.066,E2 7939.066} C_VEL
LIN {X 0,Y 601.069,Z 762.06,A -85,B 0,C 180,E1 7943.706,E2 7943.706} C_VEL
LIN {X 0,Y 601.019,Z 762.06,A -85,B 0,C 180,E1 7948.522,E2 7948.522} C_VEL
LIN {X 0,Y 600.924,Z 762.06,A -85,B 0,C 180,E1 7953.92,E2 7953.92} C_VEL
LIN {X 0,Y 600.889,Z 762.06,A -85,B 0,C 180,E1 7958.938,E2 7958.938} C_VEL
LIN {X 0,Y 600.826,Z 762.06,A -85,B 0,C 180,E1 7961.603,E2 7961.603} C_VEL
LIN {X 0,Y 603.511,Z 767.966,A -85,B 0,C 180,E1 7962.019,E2 7962.019} C_VEL
LIN {X 0,Y 629.688,Z 811.487,A -85,B 0,C 180,E1 7965.412,E2 7965.412} C_VEL
LIN {X 0,Y 637.366,Z 826.573,A -85,B 0,C 180,E1 7966.459,E2 7966.459} C_VEL
LIN {X 0,Y 633.657,Z 876.944,A -85,B 0,C 180,E1 7967.892,E2 7967.892} C_VEL
LIN {X 0,Y 629.269,Z 922.095,A -85,B 0,C 180,E1 7969.739,E2 7969.739} C_VEL
LIN {X 0,Y 624.257,Z 964.615,A -85,B 0,C 180,E1 7972.072,E2 7972.072} C_VEL
LIN {X 0,Y 618.819,Z 1007.258,A -85,B 0,C 180,E1 7975.07,E2 7975.07} C_VEL
LIN {X 0,Y 613.749,Z 1045.867,A -85,B 0,C 180,E1 7978.535,E2 7978.535} C_VEL
LIN {X 0,Y 609.507,Z 1079.663,A -85,B 0,C 180,E1 7982.3,E2 7982.3} C_VEL
LIN {X 0,Y 606.119,Z 1109.523,A -85,B 0,C 180,E1 7986.492,E2 7986.492} C_VEL
LIN {X 0,Y 603.968,Z 1133.061,A -85,B 0,C 180,E1 7990.64,E2 7990.64} C_VEL
LIN {X 0,Y 602.722,Z 1152.221,A -85,B 0,C 180,E1 7995.025,E2 7995.025} C_VEL
LIN {X 0,Y 602.103,Z 1165.528,A -85,B 0,C 180,E1 7999.151,E2 7999.151} C_VEL
LIN {X 0,Y 601.941,Z 1174.848,A -85,B 0,C 180,E1 8003.514,E2 8003.514} C_VEL
LIN {X 0,Y 601.767,Z 1178.957,A -85,B 0,C 180,E1 8007.122,E2 8007.122} C_VEL
LIN {X 0,Y 601.863,Z 1179.656,A -85,B 0,C 180,E1 8011.439,E2 8011.439} C_VEL
LIN {X 0,Y 601.933,Z 1175.846,A -85,B 0,C 180,E1 8015.764,E2 8015.764} C_VEL
LIN {X 0,Y 602.02,Z 1167.21,A -85,B 0,C 180,E1 8020.12,E2 8020.12} C_VEL
LIN {X 0,Y 602.69,Z 1153.544,A -85,B 0,C 180,E1 8024.521,E2 8024.521} C_VEL
LIN {X 0,Y 603.91,Z 1134.517,A -85,B 0,C 180,E1 8028.984,E2 8028.984} C_VEL
LIN {X 0,Y 606.28,Z 1108.961,A -85,B 0,C 180,E1 8033.503,E2 8033.503} C_VEL
LIN {X 0,Y 609.667,Z 1078.935,A -85,B 0,C 180,E1 8037.693,E2 8037.693} C_VEL
LIN {X 0,Y 614.284,Z 1041.755,A -85,B 0,C 180,E1 8041.788,E2 8041.788} C_VEL
LIN {X 0,Y 619.152,Z 1004.449,A -85,B 0,C 180,E1 8045.058,E2 8045.058} C_VEL
LIN {X 0,Y 624.803,Z 959.856,A -85,B 0,C 180,E1 8048.14,E2 8048.14} C_VEL
LIN {X 0,Y 629.928,Z 915.931,A -85,B 0,C 180,E1 8050.448,E2 8050.448} C_VEL
LIN {X 0,Y 634.13,Z 872.308,A -85,B 0,C 180,E1 8052.17,E2 8052.17} C_VEL
LIN {X 0,Y 637.247,Z 830.348,A -85,B 0,C 180,E1 8053.349,E2 8053.349} C_VEL
LIN {X 0,Y 636.465,Z 825.419,A -85,B 0,C 180,E1 8053.56,E2 8053.56} C_VEL
LIN {X 0,Y 617.518,Z 790.09,A -85,B 0,C 180,E1 8056.083,E2 8056.083} C_VEL
LIN {X 0,Y 601.208,Z 764.106,A -85,B 0,C 180,E1 8058.205,E2 8058.205} C_VEL
LIN {X 0,Y 600.942,Z 762.06,A -85,B 0,C 180,E1 8058.342,E2 8058.342} C_VEL
LIN {X 0,Y 600.896,Z 762.06,A -85,B 0,C 180,E1 8063.585,E2 8063.585} C_VEL
LIN {X 0,Y 600.922,Z 762.06,A -85,B 0,C 180,E1 8068.759,E2 8068.759} C_VEL
LIN {X 0,Y 600.96,Z 762.06,A -85,B 0,C 180,E1 8074.706,E2 8074.706} C_VEL
LIN {X 0,Y 601.001,Z 762.06,A -85,B 0,C 180,E1 8079.402,E2 8079.402} C_VEL
LIN {X 0,Y 601.187,Z 762.06,A -85,B 0,C 180,E1 8085.453,E2 8085.453} C_VEL
LIN {X 0,Y 601.457,Z 762.06,A -85,B 0,C 180,E1 8089.881,E2 8089.881} C_VEL
LIN {X 0,Y 601.594,Z 762.06,A -85,B 0,C 180,E1 8094.243,E2 8094.243} C_VEL
LIN {X 0,Y 601.764,Z 762.06,A -85,B 0,C 180,E1 8098.57,E2 8098.57} C_VEL
LIN {X 0,Y 601.662,Z 762.06,A -85,B 0,C 180,E1 8102.887,E2 8102.887} C_VEL
LIN {X 0,Y 601.519,Z 762.06,A -85,B 0,C 180,E1 8108.677,E2 8108.677} C_VEL
LIN {X 0,Y 601.388,Z 762.06,A -85,B 0,C 180,E1 8114.559,E2 8114.559} C_VEL
LIN {X 0,Y 601.357,Z 762.06,A -85,B 0,C 180,E1 8119.073,E2 8119.073} C_VEL
LIN {X 0,Y 601.201,Z 762.06,A -85,B 0,C 180,E1 8123.719,E2 8123.719} C_VEL
LIN {X 0,Y 601.122,Z 762.06,A -85,B 0,C 180,E1 8128.536,E2 8128.536} C_VEL
LIN {X 0,Y 600.963,Z 762.06,A -85,B 0,C 180,E1 8133.923,E2 8133.923} C_VEL
LIN {X 0,Y 600.925,Z 762.06,A -85,B 0,C 180,E1 8138.956,E2 8138.956} C_VEL
LIN {X 0,Y 600.96,Z 762.066,A -85,B 0,C 180,E1 8141.226,E2 8141.226} C_VEL
LIN {X 0,Y 603.297,Z 767.629,A -85,B 0,C 180,E1 8141.574,E2 8141.574} C_VEL
LIN {X 0,Y 627.721,Z 807.267,A -85,B 0,C 180,E1 8144.642,E2 8144.642} C_VEL
LIN {X 0,Y 638.858,Z 828.822,A -85,B 0,C 180,E1 8146.005,E2 8146.005} C_VEL
LIN {X 0,Y 638.156,Z 844.941,A -85,B 0,C 180,E1 8146.289,E2 8146.289} C_VEL
LIN {X 0,Y 634.33,Z 862.034,A -85,B 0,C 180,E1 8146.399,E2 8146.399} C_VEL
LIN {X 0,Y 630.038,Z 878.934,A -85,B 0,C 180,E1 8146.565,E2 8146.565} C_VEL
LIN {X 0,Y 625.733,Z 926.778,A -85,B 0,C 180,E1 8148.188,E2 8148.188} C_VEL
LIN {X 0,Y 620.626,Z 972.009,A -85,B 0,C 180,E1 8150.317,E2 8150.317} C_VEL
LIN {X 0,Y 614.526,Z 1018.342,A -85,B 0,C 180,E1 8153.231,E2 8153.231} C_VEL
LIN {X 0,Y 609.398,Z 1056.697,A -85,B 0,C 180,E1 8156.336,E2 8156.336} C_VEL
LIN {X 0,Y 604.183,Z 1094.59,A -85,B 0,C 180,E1 8160.18,E2 8160.18} C_VEL
LIN {X 0,Y 600.136,Z 1126.563,A -85,B 0,C 180,E1 8164.267,E2 8164.267} C_VEL
LIN {X 0,Y 597.104,Z 1154.989,A -85,B 0,C 180,E1 8168.86,E2 8168.86} C_VEL
LIN {X 0,Y 595.242,Z 1176.472,A -85,B 0,C 180,E1 8173.405,E2 8173.405} C_VEL
LIN {X 0,Y 594.372,Z 1191.171,A -85,B 0,C 180,E1 8177.519,E2 8177.519} C_VEL
LIN {X 0,Y 594.012,Z 1202.22,A -85,B 0,C 180,E1 8181.956,E2 8181.956} C_VEL
LIN {X 0,Y 593.884,Z 1207.676,A -85,B 0,C 180,E1 8185.621,E2 8185.621} C_VEL
LIN {X 0,Y 593.982,Z 1210,A -85,B 0,C 180,E1 8189.999,E2 8189.999} C_VEL
LIN {X 0,Y 593.883,Z 1207.678,A -85,B 0,C 180,E1 8194.377,E2 8194.377} C_VEL
LIN {X 0,Y 594.036,Z 1200.69,A -85,B 0,C 180,E1 8198.779,E2 8198.779} C_VEL
LIN {X 0,Y 594.495,Z 1188.886,A -85,B 0,C 180,E1 8203.224,E2 8203.224} C_VEL
LIN {X 0,Y 595.688,Z 1171.707,A -85,B 0,C 180,E1 8207.722,E2 8207.722} C_VEL
LIN {X 0,Y 597.726,Z 1148.504,A -85,B 0,C 180,E1 8212.284,E2 8212.284} C_VEL
LIN {X 0,Y 600.806,Z 1121.247,A -85,B 0,C 180,E1 8216.487,E2 8216.487} C_VEL
LIN {X 0,Y 605.298,Z 1086.111,A -85,B 0,C 180,E1 8220.763,E2 8220.763} C_VEL
LIN {X 0,Y 610.41,Z 1048.799,A -85,B 0,C 180,E1 8224.361,E2 8224.361} C_VEL
LIN {X 0,Y 616.191,Z 1006.73,A -85,B 0,C 180,E1 8227.576,E2 8227.576} C_VEL
LIN {X 0,Y 621.851,Z 961.941,A -85,B 0,C 180,E1 8230.204,E2 8230.204} C_VEL
LIN {X 0,Y 627.014,Z 914.627,A -85,B 0,C 180,E1 8232.289,E2 8232.289} C_VEL
LIN {X 0,Y 630.8,Z 868.828,A -85,B 0,C 180,E1 8233.693,E2 8233.693} C_VEL
LIN {X 0,Y 632.607,Z 829.88,A -85,B 0,C 180,E1 8234.521,E2 8234.521} C_VEL
LIN {X 0,Y 609.92,Z 790.274,A -85,B 0,C 180,E1 8237.35,E2 8237.35} C_VEL
LIN {X 0,Y 593.098,Z 763.364,A -85,B 0,C 180,E1 8239.619,E2 8239.619} C_VEL
LIN {X 0,Y 592.988,Z 762.06,A -85,B 0,C 180,E1 8239.741,E2 8239.741} C_VEL
LIN {X 0,Y 593.034,Z 762.06,A -85,B 0,C 180,E1 8244.625,E2 8244.625} C_VEL
LIN {X 0,Y 593.024,Z 762.06,A -85,B 0,C 180,E1 8250.038,E2 8250.038} C_VEL
LIN {X 0,Y 593.1,Z 762.06,A -85,B 0,C 180,E1 8254.328,E2 8254.328} C_VEL
LIN {X 0,Y 593.219,Z 762.06,A -85,B 0,C 180,E1 8259.101,E2 8259.101} C_VEL
LIN {X 0,Y 593.417,Z 762.06,A -85,B 0,C 180,E1 8263.727,E2 8263.727} C_VEL
LIN {X 0,Y 593.564,Z 762.06,A -85,B 0,C 180,E1 8269.727,E2 8269.727} C_VEL
LIN {X 0,Y 593.785,Z 762.06,A -85,B 0,C 180,E1 8275.613,E2 8275.613} C_VEL
LIN {X 0,Y 593.947,Z 762.06,A -85,B 0,C 180,E1 8279.992,E2 8279.992} C_VEL
LIN {X 0,Y 593.79,Z 762.06,A -85,B 0,C 180,E1 8284.37,E2 8284.37} C_VEL
LIN {X 0,Y 593.667,Z 762.06,A -85,B 0,C 180,E1 8288.775,E2 8288.775} C_VEL
LIN {X 0,Y 593.293,Z 762.06,A -85,B 0,C 180,E1 8294.57,E2 8294.57} C_VEL
LIN {X 0,Y 593.178,Z 762.06,A -85,B 0,C 180,E1 8300.883,E2 8300.883} C_VEL
LIN {X 0,Y 593.124,Z 762.06,A -85,B 0,C 180,E1 8305.652,E2 8305.652} C_VEL
LIN {X 0,Y 593.078,Z 762.06,A -85,B 0,C 180,E1 8310.622,E2 8310.622} C_VEL
LIN {X 0,Y 593.007,Z 762.06,A -85,B 0,C 180,E1 8315.864,E2 8315.864} C_VEL
LIN {X 0,Y 592.943,Z 762.805,A -85,B 0,C 180,E1 8320.77,E2 8320.77} C_VEL
LIN {X 0,Y 595.836,Z 768.206,A -85,B 0,C 180,E1 8321.192,E2 8321.192} C_VEL
LIN {X 0,Y 621.847,Z 811.162,A -85,B 0,C 180,E1 8324.679,E2 8324.679} C_VEL
LIN {X 0,Y 631.361,Z 830.152,A -85,B 0,C 180,E1 8326.046,E2 8326.046} C_VEL
LIN {X 0,Y 627.226,Z 882.191,A -85,B 0,C 180,E1 8327.58,E2 8327.58} C_VEL
LIN {X 0,Y 622.497,Z 926.886,A -85,B 0,C 180,E1 8329.498,E2 8329.498} C_VEL
LIN {X 0,Y 616.72,Z 973.097,A -85,B 0,C 180,E1 8332.143,E2 8332.143} C_VEL
LIN {X 0,Y 611.236,Z 1013.152,A -85,B 0,C 180,E1 8335.118,E2 8335.118} C_VEL
LIN {X 0,Y 605.853,Z 1052.179,A -85,B 0,C 180,E1 8338.769,E2 8338.769} C_VEL
LIN {X 0,Y 601.278,Z 1086.602,A -85,B 0,C 180,E1 8342.847,E2 8342.847} C_VEL
LIN {X 0,Y 598.107,Z 1114.842,A -85,B 0,C 180,E1 8347.034,E2 8347.034} C_VEL
LIN {X 0,Y 595.903,Z 1138.411,A -85,B 0,C 180,E1 8351.513,E2 8351.513} C_VEL
LIN {X 0,Y 594.745,Z 1156.541,A -85,B 0,C 180,E1 8356.033,E2 8356.033} C_VEL
LIN {X 0,Y 594.127,Z 1169.207,A -85,B 0,C 180,E1 8360.485,E2 8360.485} C_VEL
LIN {X 0,Y 593.966,Z 1175.969,A -85,B 0,C 180,E1 8364.16,E2 8364.16} C_VEL
LIN {X 0,Y 593.787,Z 1179.678,A -85,B 0,C 180,E1 8368.542,E2 8368.542} C_VEL
LIN {X 0,Y 593.866,Z 1178.889,A -85,B 0,C 180,E1 8372.918,E2 8372.918} C_VEL
LIN {X 0,Y 594.041,Z 1173.43,A -85,B 0,C 180,E1 8377.341,E2 8377.341} C_VEL
LIN {X 0,Y 594.386,Z 1163.285,A -85,B 0,C 180,E1 8381.736,E2 8381.736} C_VEL
LIN {X 0,Y 595.239,Z 1147.82,A -85,B 0,C 180,E1 8386.216,E2 8386.216} C_VEL
LIN {X 0,Y 596.919,Z 1126.739,A -85,B 0,C 180,E1 8390.758,E2 8390.758} C_VEL
LIN {X 0,Y 599.611,Z 1100.91,A -85,B 0,C 180,E1 8395.056,E2 8395.056} C_VEL
LIN {X 0,Y 603.652,Z 1068.692,A -85,B 0,C 180,E1 8399.303,E2 8399.303} C_VEL
LIN {X 0,Y 608.397,Z 1033.554,A -85,B 0,C 180,E1 8402.985,E2 8402.985} C_VEL
LIN {X 0,Y 614.157,Z 992.458,A -85,B 0,C 180,E1 8406.42,E2 8406.42} C_VEL
LIN {X 0,Y 619.76,Z 949.519,A -85,B 0,C 180,E1 8409.204,E2 8409.204} C_VEL
LIN {X 0,Y 625.102,Z 902.841,A -85,B 0,C 180,E1 8411.529,E2 8411.529} C_VEL
LIN {X 0,Y 629.712,Z 852.555,A -85,B 0,C 180,E1 8413.288,E2 8413.288} C_VEL
LIN {X 0,Y 630.95,Z 829.538,A -85,B 0,C 180,E1 8413.919,E2 8413.919} C_VEL
LIN {X 0,Y 611.883,Z 793.642,A -85,B 0,C 180,E1 8416.569,E2 8416.569} C_VEL
LIN {X 0,Y 593.115,Z 763.479,A -85,B 0,C 180,E1 8419.107,E2 8419.107} C_VEL
LIN {X 0,Y 592.997,Z 762.06,A -85,B 0,C 180,E1 8419.229,E2 8419.229} C_VEL
LIN {X 0,Y 592.997,Z 762.06,A -85,B 0,C 180,E1 8424.632,E2 8424.632} C_VEL
LIN {X 0,Y 592.978,Z 762.06,A -85,B 0,C 180,E1 8430.049,E2 8430.049} C_VEL
LIN {X 0,Y 593.014,Z 762.06,A -85,B 0,C 180,E1 8434.343,E2 8434.343} C_VEL
LIN {X 0,Y 593.113,Z 762.06,A -85,B 0,C 180,E1 8439.115,E2 8439.115} C_VEL
LIN {X 0,Y 593.309,Z 762.06,A -85,B 0,C 180,E1 8445.43,E2 8445.43} C_VEL
LIN {X 0,Y 593.682,Z 762.06,A -85,B 0,C 180,E1 8451.225,E2 8451.225} C_VEL
LIN {X 0,Y 593.922,Z 762.06,A -85,B 0,C 180,E1 8457.092,E2 8457.092} C_VEL
LIN {X 0,Y 593.936,Z 762.06,A -85,B 0,C 180,E1 8461.466,E2 8461.466} C_VEL
LIN {X 0,Y 593.663,Z 762.06,A -85,B 0,C 180,E1 8467.319,E2 8467.319} C_VEL
LIN {X 0,Y 593.502,Z 762.06,A -85,B 0,C 180,E1 8471.76,E2 8471.76} C_VEL
LIN {X 0,Y 593.471,Z 762.06,A -85,B 0,C 180,E1 8476.272,E2 8476.272} C_VEL
LIN {X 0,Y 593.37,Z 762.06,A -85,B 0,C 180,E1 8480.894,E2 8480.894} C_VEL
LIN {X 0,Y 593.241,Z 762.06,A -85,B 0,C 180,E1 8485.666,E2 8485.666} C_VEL
LIN {X 0,Y 593.15,Z 762.06,A -85,B 0,C 180,E1 8490.637,E2 8490.637} C_VEL
LIN {X 0,Y 593.036,Z 762.06,A -85,B 0,C 180,E1 8495.883,E2 8495.883} C_VEL
LIN {X 0,Y 592.98,Z 762.101,A -85,B 0,C 180,E1 8500.346,E2 8500.346} C_VEL
LIN {X 0,Y 595.195,Z 767.505,A -85,B 0,C 180,E1 8500.692,E2 8500.692} C_VEL
LIN {X 0,Y 618.107,Z 803.905,A -85,B 0,C 180,E1 8503.685,E2 8503.685} C_VEL
LIN {X 0,Y 632.991,Z 830.48,A -85,B 0,C 180,E1 8505.524,E2 8505.524} C_VEL
LIN {X 0,Y 630.038,Z 878.934,A -85,B 0,C 180,E1 8506.565,E2 8506.565} C_VEL
LIN {X 0,Y 625.604,Z 896.308,A -85,B 0,C 180,E1 8506.82,E2 8506.82} C_VEL
LIN {X 0,Y 621.242,Z 912.315,A -85,B 0,C 180,E1 8507.127,E2 8507.127} C_VEL
LIN {X 0,Y 616.295,Z 957.546,A -85,B 0,C 180,E1 8509.09,E2 8509.09} C_VEL
LIN {X 0,Y 610.415,Z 1002.468,A -85,B 0,C 180,E1 8511.681,E2 8511.681} C_VEL
LIN {X 0,Y 604.775,Z 1041.409,A -85,B 0,C 180,E1 8514.571,E2 8514.571} C_VEL
LIN {X 0,Y 598.825,Z 1081.929,A -85,B 0,C 180,E1 8518.378,E2 8518.378} C_VEL
LIN {X 0,Y 594.062,Z 1115.209,A -85,B 0,C 180,E1 8522.339,E2 8522.339} C_VEL
LIN {X 0,Y 590.493,Z 1144.737,A -85,B 0,C 180,E1 8526.747,E2 8526.747} C_VEL
LIN {X 0,Y 588.157,Z 1168.238,A -85,B 0,C 180,E1 8531.267,E2 8531.267} C_VEL
LIN {X 0,Y 586.933,Z 1186.373,A -85,B 0,C 180,E1 8535.842,E2 8535.842} C_VEL
LIN {X 0,Y 586.284,Z 1199.103,A -85,B 0,C 180,E1 8540.355,E2 8540.355} C_VEL
LIN {X 0,Y 586.085,Z 1205.909,A -85,B 0,C 180,E1 8544.08,E2 8544.08} C_VEL
LIN {X 0,Y 585.967,Z 1209.667,A -85,B 0,C 180,E1 8548.522,E2 8548.522} C_VEL
LIN {X 0,Y 586.098,Z 1208.919,A -85,B 0,C 180,E1 8552.955,E2 8552.955} C_VEL
LIN {X 0,Y 586.109,Z 1203.56,A -85,B 0,C 180,E1 8557.406,E2 8557.406} C_VEL
LIN {X 0,Y 586.451,Z 1193.421,A -85,B 0,C 180,E1 8561.895,E2 8561.895} C_VEL
LIN {X 0,Y 587.316,Z 1178.007,A -85,B 0,C 180,E1 8566.44,E2 8566.44} C_VEL
LIN {X 0,Y 589.189,Z 1156.973,A -85,B 0,C 180,E1 8571.042,E2 8571.042} C_VEL
LIN {X 0,Y 592.077,Z 1131.458,A -85,B 0,C 180,E1 8575.359,E2 8575.359} C_VEL
LIN {X 0,Y 596.578,Z 1098.101,A -85,B 0,C 180,E1 8579.807,E2 8579.807} C_VEL
LIN {X 0,Y 601.755,Z 1061.513,A -85,B 0,C 180,E1 8583.653,E2 8583.653} C_VEL
LIN {X 0,Y 607.694,Z 1021.068,A -85,B 0,C 180,E1 8587.032,E2 8587.032} C_VEL
LIN {X 0,Y 613.888,Z 976.626,A -85,B 0,C 180,E1 8589.893,E2 8589.893} C_VEL
LIN {X 0,Y 619.169,Z 933.887,A -85,B 0,C 180,E1 8592.008,E2 8592.008} C_VEL
LIN {X 0,Y 623.309,Z 890.819,A -85,B 0,C 180,E1 8593.581,E2 8593.581} C_VEL
LIN {X 0,Y 626.627,Z 844.179,A -85,B 0,C 180,E1 8594.736,E2 8594.736} C_VEL
LIN {X 0,Y 626.685,Z 832.885,A -85,B 0,C 180,E1 8594.995,E2 8594.995} C_VEL
LIN {X 0,Y 604.737,Z 794.507,A -85,B 0,C 180,E1 8597.809,E2 8597.809} C_VEL
LIN {X 0,Y 586.962,Z 767.205,A -85,B 0,C 180,E1 8600.251,E2 8600.251} C_VEL
LIN {X 0,Y 585.05,Z 762.06,A -85,B 0,C 180,E1 8600.583,E2 8600.583} C_VEL
LIN {X 0,Y 585.083,Z 762.06,A -85,B 0,C 180,E1 8605.737,E2 8605.737} C_VEL
LIN {X 0,Y 585.1,Z 762.06,A -85,B 0,C 180,E1 8611.413,E2 8611.413} C_VEL
LIN {X 0,Y 585.235,Z 762.06,A -85,B 0,C 180,E1 8617.207,E2 8617.207} C_VEL
LIN {X 0,Y 585.426,Z 762.06,A -85,B 0,C 180,E1 8622.753,E2 8622.753} C_VEL
LIN {X 0,Y 585.616,Z 762.06,A -85,B 0,C 180,E1 8628.675,E2 8628.675} C_VEL
LIN {X 0,Y 585.824,Z 762.06,A -85,B 0,C 180,E1 8634.07,E2 8634.07} C_VEL
LIN {X 0,Y 586.06,Z 762.06,A -85,B 0,C 180,E1 8639.991,E2 8639.991} C_VEL
LIN {X 0,Y 585.899,Z 762.06,A -85,B 0,C 180,E1 8644.428,E2 8644.428} C_VEL
LIN {X 0,Y 585.742,Z 762.06,A -85,B 0,C 180,E1 8648.895,E2 8648.895} C_VEL
LIN {X 0,Y 585.432,Z 762.06,A -85,B 0,C 180,E1 8653.422,E2 8653.422} C_VEL
LIN {X 0,Y 585.219,Z 762.06,A -85,B 0,C 180,E1 8659.602,E2 8659.602} C_VEL
LIN {X 0,Y 585.195,Z 762.06,A -85,B 0,C 180,E1 8665.342,E2 8665.342} C_VEL
LIN {X 0,Y 585.113,Z 762.06,A -85,B 0,C 180,E1 8671.085,E2 8671.085} C_VEL
LIN {X 0,Y 585.007,Z 762.06,A -85,B 0,C 180,E1 8676.799,E2 8676.799} C_VEL
LIN {X 0,Y 584.986,Z 762.172,A -85,B 0,C 180,E1 8679.84,E2 8679.84} C_VEL
LIN {X 0,Y 587.375,Z 767.729,A -85,B 0,C 180,E1 8680.224,E2 8680.224} C_VEL
LIN {X 0,Y 610.289,Z 804.19,A -85,B 0,C 180,E1 8683.392,E2 8683.392} C_VEL
LIN {X 0,Y 625.453,Z 833.132,A -85,B 0,C 180,E1 8685.607,E2 8685.607} C_VEL
LIN {X 0,Y 621.178,Z 883.968,A -85,B 0,C 180,E1 8687.142,E2 8687.142} C_VEL
LIN {X 0,Y 615.84,Z 930.69,A -85,B 0,C 180,E1 8689.201,E2 8689.201} C_VEL
LIN {X 0,Y 610.003,Z 975.269,A -85,B 0,C 180,E1 8691.814,E2 8691.814} C_VEL
LIN {X 0,Y 604.141,Z 1015.586,A -85,B 0,C 180,E1 8694.881,E2 8694.881} C_VEL
LIN {X 0,Y 598.532,Z 1053.923,A -85,B 0,C 180,E1 8698.543,E2 8698.543} C_VEL
LIN {X 0,Y 593.649,Z 1088.452,A -85,B 0,C 180,E1 8702.731,E2 8702.731} C_VEL
LIN {X 0,Y 590.384,Z 1116.019,A -85,B 0,C 180,E1 8706.929,E2 8706.929} C_VEL
LIN {X 0,Y 588.005,Z 1140.348,A -85,B 0,C 180,E1 8711.69,E2 8711.69} C_VEL
LIN {X 0,Y 586.847,Z 1157.828,A -85,B 0,C 180,E1 8716.221,E2 8716.221} C_VEL
LIN {X 0,Y 586.155,Z 1170.781,A -85,B 0,C 180,E1 8721.102,E2 8721.102} C_VEL
LIN {X 0,Y 586.082,Z 1175.969,A -85,B 0,C 180,E1 8724.081,E2 8724.081} C_VEL
LIN {X 0,Y 585.886,Z 1179.678,A -85,B 0,C 180,E1 8728.523,E2 8728.523} C_VEL
LIN {X 0,Y 585.963,Z 1178.886,A -85,B 0,C 180,E1 8732.957,E2 8732.957} C_VEL
LIN {X 0,Y 586.173,Z 1173.484,A -85,B 0,C 180,E1 8737.407,E2 8737.407} C_VEL
LIN {X 0,Y 586.527,Z 1163.286,A -85,B 0,C 180,E1 8741.895,E2 8741.895} C_VEL
LIN {X 0,Y 587.439,Z 1147.821,A -85,B 0,C 180,E1 8746.438,E2 8746.438} C_VEL
LIN {X 0,Y 589.228,Z 1126.744,A -85,B 0,C 180,E1 8751.042,E2 8751.042} C_VEL
LIN {X 0,Y 592.127,Z 1100.91,A -85,B 0,C 180,E1 8755.396,E2 8755.396} C_VEL
LIN {X 0,Y 596.594,Z 1067.741,A -85,B 0,C 180,E1 8759.808,E2 8759.808} C_VEL
LIN {X 0,Y 601.894,Z 1030.888,A -85,B 0,C 180,E1 8763.663,E2 8763.663} C_VEL
LIN {X 0,Y 607.743,Z 991.483,A -85,B 0,C 180,E1 8766.949,E2 8766.949} C_VEL
LIN {X 0,Y 613.533,Z 949.097,A -85,B 0,C 180,E1 8769.709,E2 8769.709} C_VEL
LIN {X 0,Y 619.133,Z 902.854,A -85,B 0,C 180,E1 8772.02,E2 8772.02} C_VEL
LIN {X 0,Y 624.005,Z 852.114,A -85,B 0,C 180,E1 8773.809,E2 8773.809} C_VEL
LIN {X 0,Y 624.999,Z 832.652,A -85,B 0,C 180,E1 8774.36,E2 8774.36} C_VEL
LIN {X 0,Y 606.13,Z 796.718,A -85,B 0,C 180,E1 8777.09,E2 8777.09} C_VEL
LIN {X 0,Y 586.979,Z 767.239,A -85,B 0,C 180,E1 8779.74,E2 8779.74} C_VEL
LIN {X 0,Y 585.055,Z 762.06,A -85,B 0,C 180,E1 8780.131,E2 8780.131} C_VEL
LIN {X 0,Y 585.072,Z 762.06,A -85,B 0,C 180,E1 8785.741,E2 8785.741} C_VEL
LIN {X 0,Y 585.038,Z 762.06,A -85,B 0,C 180,E1 8791.427,E2 8791.427} C_VEL
LIN {X 0,Y 585.139,Z 762.06,A -85,B 0,C 180,E1 8797.221,E2 8797.221} C_VEL
LIN {X 0,Y 585.198,Z 762.06,A -85,B 0,C 180,E1 8802.83,E2 8802.83} C_VEL
LIN {X 0,Y 585.568,Z 762.06,A -85,B 0,C 180,E1 8808.706,E2 8808.706} C_VEL
LIN {X 0,Y 585.811,Z 762.06,A -85,B 0,C 180,E1 8814.087,E2 8814.087} C_VEL
LIN {X 0,Y 585.962,Z 762.06,A -85,B 0,C 180,E1 8818.531,E2 8818.531} C_VEL
LIN {X 0,Y 585.857,Z 762.06,A -85,B 0,C 180,E1 8822.965,E2 8822.965} C_VEL
LIN {X 0,Y 585.747,Z 762.06,A -85,B 0,C 180,E1 8827.419,E2 8827.419} C_VEL
LIN {X 0,Y 585.571,Z 762.06,A -85,B 0,C 180,E1 8833.437,E2 8833.437} C_VEL
LIN {X 0,Y 585.55,Z 762.06,A -85,B 0,C 180,E1 8838.047,E2 8838.047} C_VEL
LIN {X 0,Y 585.379,Z 762.06,A -85,B 0,C 180,E1 8842.788,E2 8842.788} C_VEL
LIN {X 0,Y 585.248,Z 762.06,A -85,B 0,C 180,E1 8848.611,E2 8848.611} C_VEL
LIN {X 0,Y 585.144,Z 762.06,A -85,B 0,C 180,E1 8854.626,E2 8854.626} C_VEL
LIN {X 0,Y 585.09,Z 762.631,A -85,B 0,C 180,E1 8859.446,E2 8859.446} C_VEL
LIN {X 0,Y 587.803,Z 768.013,A -85,B 0,C 180,E1 8859.864,E2 8859.864} C_VEL
LIN {X 0,Y 612.588,Z 807.292,A -85,B 0,C 180,E1 8863.203,E2 8863.203} C_VEL
LIN {X 0,Y 627.238,Z 833.865,A -85,B 0,C 180,E1 8865.074,E2 8865.074} C_VEL
LIN {X 0,Y 623.798,Z 883.589,A -85,B 0,C 180,E1 8866.198,E2 8866.198} C_VEL
LIN {X 0,Y 621.242,Z 912.315,A -85,B 0,C 180,E1 8867.127,E2 8867.127} C_VEL
LIN {X 0,Y 616.606,Z 928.719,A -85,B 0,C 180,E1 8867.516,E2 8867.516} C_VEL
LIN {X 0,Y 611.803,Z 944.782,A -85,B 0,C 180,E1 8867.982,E2 8867.982} C_VEL
LIN {X 0,Y 606.227,Z 987.494,A -85,B 0,C 180,E1 8870.246,E2 8870.246} C_VEL
LIN {X 0,Y 599.817,Z 1029.525,A -85,B 0,C 180,E1 8873.151,E2 8873.151} C_VEL
LIN {X 0,Y 593.92,Z 1068.261,A -85,B 0,C 180,E1 8876.549,E2 8876.549} C_VEL
LIN {X 0,Y 588.34,Z 1104.494,A -85,B 0,C 180,E1 8880.579,E2 8880.579} C_VEL
LIN {X 0,Y 584.077,Z 1135.391,A -85,B 0,C 180,E1 8884.897,E2 8884.897} C_VEL
LIN {X 0,Y 581.083,Z 1161.254,A -85,B 0,C 180,E1 8889.524,E2 8889.524} C_VEL
LIN {X 0,Y 579.347,Z 1181.009,A -85,B 0,C 180,E1 8894.104,E2 8894.104} C_VEL
LIN {X 0,Y 578.567,Z 1194.284,A -85,B 0,C 180,E1 8898.265,E2 8898.265} C_VEL
LIN {X 0,Y 578.225,Z 1203.554,A -85,B 0,C 180,E1 8902.491,E2 8902.491} C_VEL
